# B&R Automation Studio project Palletizer
Automation Studio 4.10.2.37; technology packages: Acp10Arnc0 5.20.2, mappView 5.20.0

## Configuration Default_Config

CPU X20CP1382, AutomationRuntime A4.83, Build 4.1.2, Safety 0.0, Vc V4.72.3

### Hardware
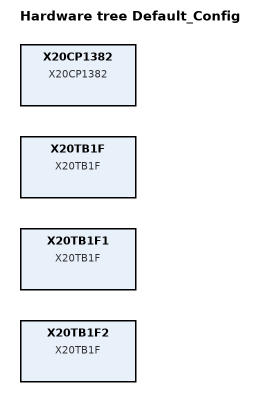
```
X20CP1382 : X20CP1382 v1.14.0.0  [X1 -> X1.SL; X2 -> X2.SL; X3 -> X3.SL]
  Module X1 (Type=X1, Virtual=true, Version=1.14.0.0)
    Connection (Connector=SS1, TargetModule=X20TB1F, TargetConnector=SS)
    Connection (Connector=SL, TargetModule=X20CP1382, TargetConnector=X1)
  Module X2 (Type=X2, Virtual=true, Version=1.14.0.0)
    Connection (Connector=SS1, TargetModule=X20TB1F1, TargetConnector=SS)
    Connection (Connector=SL, TargetModule=X20CP1382, TargetConnector=X2)
  Module X3 (Type=X3, Virtual=true, Version=1.14.0.0)
    Connection (Connector=SS1, TargetModule=X20TB1F2, TargetConnector=SS)
    Connection (Connector=SL, TargetModule=X20CP1382, TargetConnector=X3)
  Connector IF2:
    ActivateDevice = 1
    Vnc1
    VncKeyMappingFile1 = 
    VncRefreshRate1 = 100
  Connector IF3:
    DNAConfiguration = manual
    CycleTime = 2000
  ConfigurationID = Palletizer_Default_Config
  Simulation = 1
  Cyclic1Tolerance = 0
  Cyclic2Tolerance = 0
  TimeZone = 140
  ActivateOpcUa = 1
  OpcUaInformationModels_PV_Version = 1
X20TB1F : X20TB1F v1.0.0.0
X20TB1F1 : X20TB1F v1.0.0.0
X20TB1F2 : X20TB1F v1.0.0.0
```

### Acp10cfg.ncc - X20CP1382/Motion/Acp10cfg.ncc
```
NcConfiguration (Version=5.06.2, NcSwId=Acp10)
  ACP10CF1_typ:
    cnt_nettrc_rec_drive = 150
    bufsize_trace_upload = 1200
    tc_nc_man_task = Cyclic #1
    glob_pv_as_ncobject = Yes
    ncsys_dl_broadcast = Yes
    ncsys_dl_acp_reset = Yes
    safemc_log_err_to_ax = Yes
    network_init:
      ncsw_init_execute = Yes
      automatic_execute = No
      node_nr_warning = Yes
      net_err_before_ncact = Yes
    nettrc:
      enter_parsecrec = Yes
      enter_ncaction = Yes
      save_ring_startidx = No
    cam_prof_download:
      cam_dat_dl_parallel = No
      tc_cam_dl_parallel = Task class for NC Manager task
```

## Logical view

Binary libraries used (declarations not repeated): operator, runtime, astime, AsIecCon, standard, AsArLog, AsBrStr, AsTCP, MTBasics 2.21.0, brsystem, MTTypes 1.03.4, sys_lib, Acp10man 5.20.2, Acp10par 5.20.2, NcGlobal 5.20.2, Acp10sim 5.20.2

### Global.var - Global variables
```iecst
(*Sensors*)
VAR
	LightBarrier1 : BOOL;
	LightBarrier2 : BOOL;
	LaserSensor1 : BOOL;
	LaserSensor2 : BOOL;
END_VAR
(*Simulation variables*)
VAR
	Pusher_BKW : BOOL;
	Pusher_FWD : BOOL;
	Turnpusher_FWD : BOOL;
	Turnpusher_BWD : BOOL;
	Crane_Vacuum : BOOL;
	Pallet_ForkFB : BOOL;
	Feeder_ConveyorIF_Fwd : BOOL;
	Feeder_ConveyorTurn1_Fwd : BOOL;
	Feeder_PusherFwd : BOOL;
	Feeder_ConveyorEndFwd : BOOL;
	Feeder_TurnpusherFwd : BOOL;
	Feeder_TurnpusherBwd : BOOL;
	Crane_VacuumGrip : BOOL;
	Crane_CartboardTrig : BOOL;
	Crane_SlideRail_EN : BOOL;
	Crane_PusherZ_EN : BOOL;
	Crane_PusherX_EN : BOOL;
	Pallet_Fork_EN : BOOL;
	Pallet_Conveyor1_Fwd : BOOL;
	Feeder_Carriage_Axis : REAL;
	Feeder_Carriage_Reached : BOOL;
	Crane_Box_Axis : REAL;
	Crane_Gantry_Axis : REAL;
	Pallet_Lifter_Axis : REAL;
	Crane_Box_Axis_TgtPos : REAL;
	Feeder_Carriage_Axis_TgtPos : REAL;
	Crane_Gantry_Axis_TgtPos : REAL;
	Pallet_Conveyor2_ActVel : REAL;
	Pallet_Lifter_Axis_TgtPos : REAL;
END_VAR
(*Variables*)
VAR
	OperationType : INT := 0;
END_VAR
(*Faults*)
VAR
	OutOfPallet : BOOL;
	OutOfCartboard : BOOL;
	EmergencyStop : BOOL;
	Feeder_EmergencyStop : BOOL := FALSE;
	Crane_EmergencyStop : BOOL := FALSE;
	Pallet_EmergencyStop : BOOL := FALSE;
	Feeder_ResetConfig : BOOL := FALSE;
	Crane_ResetConfig : BOOL := FALSE;
	Pallet_ResetConfig : BOOL := FALSE;
	EnableMachine : BOOL := FALSE;
	Feeder_ImmediateStop : BOOL;
	Crane_ImmediateStop : BOOL;
	Pallet_ImmediateStop : BOOL;
	Feeder_Restart : BOOL := FALSE;
	Crane_Restart : BOOL := FALSE;
	Pallet_Restart : BOOL := FALSE;
	Feeder_OnPhaseStop : BOOL := FALSE;
	Crane_OnPhaseStop : BOOL := FALSE;
	Pallet_OnPhaseStop : BOOL := FALSE;
	ImmediateStop : BOOL;
	OnPhaseStop : BOOL;
	act_PalletConveyor2Fault : BOOL := FALSE;
	act_CartboardFault : BOOL := FALSE;
	act_CarriageFault : BOOL := FALSE;
	act_GantryCraneFault : BOOL := FALSE;
	act_BoxCraneFault : BOOL := FALSE;
	act_PalletForkFault : BOOL := FALSE;
	act_PalletLifterFault : BOOL := FALSE;
	act_FeederPusherFault : BOOL := FALSE;
	act_PusherXFault : BOOL := FALSE;
	act_PusherZFault : BOOL := FALSE;
	act_TurnpusherFault : BOOL := FALSE;
	act_SlideRailFault : BOOL := FALSE;
	act_ConveyorIFFault : BOOL := FALSE;
	act_ConveyorEndFault : BOOL := FALSE;
	act_PalletConveyor1Fault : BOOL := FALSE;
	act_ConveyorTurn1Fault : BOOL := FALSE;
	act_VacuumFault : BOOL := FALSE;
END_VAR
(*GenericDevices*)
VAR
	Conveyor_if_enable_request : BOOL;
	Conveyor_if_disable_request : BOOL;
	Conveyor_turn1_enable_request : BOOL;
	Conveyor_turn1_disable_request : BOOL;
	Pusher_enable_request : BOOL;
	Pusher_disable_request : BOOL;
	Conveyor_end_enable_request : BOOL;
	Conveyor_end_disable_request : BOOL;
	Turnpusher_enable_request : BOOL;
	Turnpusher_disable_request : BOOL;
	Vacuum_enable_request : BOOL;
	Vacuum_disable_request : BOOL;
	Cartboard_enable_request : BOOL;
	Cartboard_disable_request : BOOL;
	SlideRail_enable_request : BOOL;
	SlideRail_disable_request : BOOL;
	PusherZ_enable_request : BOOL;
	PusherZ_disable_request : BOOL;
	PusherX_enable_request : BOOL;
	PusherX_disable_request : BOOL;
	PalletFork_enable_request : BOOL;
	PalletFork_disable_request : BOOL;
	PalletConveyor1_enable_request : BOOL;
	PalletConveyor1_disable_request : BOOL;
END_VAR
(*Comunication between PALLET HANDLER and MAIN*)
VAR
	StartPallet : BOOL := FALSE; (*if TRUE the pallet handler goes to the idle state, ready to free a pallet*)
	PalletCounter : INT := 5; (*Number of pallets that are still available before a refill*)
END_VAR
(*Comunication between CRANE HANDLER and MAIN*)
VAR
	StartCrane : BOOL := FALSE; (*if TRUE the crane handler goes to the idle state, ready to receive the box layer*)
	CraneCartboardCounter : INT := 28;
END_VAR
(*Comunication between FEEDER_HANDLER and MAIN*)
VAR
	StartFeeder : BOOL := FALSE;
	CraneLayerCounter : BOOL := FALSE; (*If TRUE the feeder is working on the second layer*)
	BoxCounter : INT := 0;
END_VAR
(*MAIN*)
VAR
	StartMachine : BOOL; (*if TRUE the machine stars*)
	CraneReady : BOOL; (*if TRUE the crane is ready to receive the boxes*)
	FeederReady : BOOL; (*if TRUE the 14 boxes are ready to be loaded on the crane*)
	LoadBoxesOnCrane : BOOL; (*if TRUE the boxes can be loaded on the crane by the feeder*)
	BoxesOnCrane : BOOL; (*if TRUE the boxes are ready to be held by the crane*)
	HoldBoxes : BOOL; (*if TRUE boxes are held by the crane*)
	PalletReady : BOOL; (*if TRUE the pallet is in position*)
	LoadBoxesOnPallet : BOOL; (*if TRUE the boxes will be loaded on the pallet*)
	SecondLayer : BOOL; (*if TRUE the feeder has finished the second layer*)
	BoxesOnPallet : BOOL; (*if TRUE the boxes are on the pallet*)
	PalletExit_EN : BOOL; (*if TRUE the pallet can move to the next station*)
	PalletExit_DONE : BOOL; (*if TRUE the pallet has gone to the next station*)
	SIMConveyorIFFault : BOOL := FALSE;
	SIMConveyorTurn1Fault : BOOL := FALSE;
	SIMFeederPusherFault : BOOL := FALSE;
	SIMConveyorEndFault : BOOL := FALSE;
	SIMTurnpusherFault : BOOL := FALSE;
	SIMCarriageFault : BOOL := FALSE;
	SIMVacuumFault : BOOL := FALSE;
	SIMSlideRailFault : BOOL := FALSE;
	SIMPusherZFault : BOOL := FALSE;
	SIMPusherXFault : BOOL := FALSE;
	SIMGantryCraneFault : BOOL := FALSE;
	SIMBoxCraneFault : BOOL := FALSE;
	SIMPalletForkFault : BOOL := FALSE;
	SIMPalletConveyor1Fault : BOOL := FALSE;
	SIMPalletLifterFault : BOOL := FALSE;
	SIMCartboardFault : BOOL := FALSE;
	SIMPalletConveyor2Fault : BOOL := FALSE;
END_VAR
(**)
VAR
	OutOfMaterial : BOOL;
END_VAR
```

### MNG_Global.typ - Global data types
```iecst
(* 3d position *)
(* position and orientation as an euler based pose *)
(* position and orientation as a 4x4 matrix *)

TYPE
	VEC3 : 	STRUCT
		x : REAL;
		y : REAL;
		z : REAL;
	END_STRUCT;
	POSE6 : 	STRUCT
		x : REAL;
		y : REAL;
		z : REAL;
		a : REAL;
		b : REAL;
		c : REAL;
	END_STRUCT;
	TRAFO : 	STRUCT
		baseX : VEC3;
		fill0 : REAL;
		baseY : VEC3;
		fill1 : REAL;
		baseZ : VEC3;
		fill2 : REAL;
		origin : VEC3;
		fill3 : REAL;
	END_STRUCT;
END_TYPE
```

### MNG_Package.typ
```iecst
(*                                                                            *)
(* File generated by the B&R AS 4 control config generator                    *)
(*                                                                            *)
(*     Provider: machineering                                                 *)
(*  Application: industrialPhysics_2.4.master                                 *)
(* Architecture: Windows 64 Bit                                               *)
(*      Version: 2.4.10491.master                                             *)
(*        Build: 164f85bec                                                    *)
(*         Date: 2020-05-19, Time: 12:11:21                                   *)
(*                                                                            *)

TYPE
	ComTCP_INPUTS_32BIT : 	STRUCT
		NumSignals : INT := 15;
		laser_sensor_IR : BOOL := 0; (* BOOL laser_sensor_IR *)
		laser_sensor2_IR : BOOL := 0; (* BOOL laser_sensor2_IR *)
		carriage_2_AXIS : REAL := 0.0; (* REAL carriage_2_AXIS *)
		carriage_2_RCHD : BOOL := 0; (* BOOL carriage_2_RCHD *)
		turnpusher_LBK : BOOL := 0; (* BOOL turnpusher_LBK *)
		turnpusher_LFR : BOOL := 0; (* BOOL turnpusher_LFR *)
		gantry_crane_AXIS : REAL := 0.0; (* REAL gantry_crane_AXIS *)
		box_crane_AXIS : REAL := 0.0; (* REAL box_crane_AXIS *)
		vaccum_box_crane_VACUUM : BOOL := 0; (* BOOL vaccum_box_crane_VACUUM *)
		pallet_light_barrier_1_IR : BOOL := 0; (* BOOL pallet_light_barrier_1_IR *)
		pallet_light_barrier_2_IR : BOOL := 0; (* BOOL pallet_light_barrier_2_IR *)
		pusher_LBK : BOOL := 0; (* BOOL pusher_LBK *)
		pusher_LFR : BOOL := 0; (* BOOL pusher_LFR *)
		pallet_lifter_AXIS : REAL := 0.0; (* REAL pallet_lifter_AXIS *)
		pallet_fork_left_FB : BOOL := 0; (* BOOL pallet_fork_left_FB *)
	END_STRUCT;
	ComTCP_OUTPUTS_32BIT : 	STRUCT
		NumSignals : INT := 18;
		cartboard_TRIG : BOOL := 0; (* BOOL cartboard_TRIG *)
		conveyor_if_FWD : BOOL := 0; (* BOOL conveyor_if_FWD *)
		conveyer_turn1_FWD : BOOL := 0; (* BOOL conveyer_turn1_FWD *)
		conveyer_end_FWD : BOOL := 0; (* BOOL conveyer_end_FWD *)
		carriage_2_TGT_POS : REAL := 0.0; (* REAL carriage_2_TGT_POS *)
		turnpusher_FWD : BOOL := 0; (* BOOL turnpusher_FWD *)
		turnpusher_BWD : BOOL := 0; (* BOOL turnpusher_BWD *)
		gantry_crane_TGT_POS : REAL := 0.0; (* REAL gantry_crane_TGT_POS *)
		box_crane_TGT_POS : REAL := 0.0; (* REAL box_crane_TGT_POS *)
		slide_rail_right_EN : BOOL := 0; (* BOOL slide_rail_right_EN *)
		vaccum_box_crane_GRIP : BOOL := 0; (* BOOL vaccum_box_crane_GRIP *)
		pusher_z_EN : BOOL := 0; (* BOOL pusher_z_EN *)
		pusher_x_EN : BOOL := 0; (* BOOL pusher_x_EN *)
		pallet_conveyor_2_ACT_VEL : REAL := 0.0; (* REAL pallet_conveyor_2_ACT_VEL *)
		pusher_FW : BOOL := 0; (* BOOL pusher_FW *)
		pallet_lifter_TGT_POS : REAL := 0.0; (* REAL pallet_lifter_TGT_POS *)
		pallet_fork_left_EN : BOOL := 0; (* BOOL pallet_fork_left_EN *)
		pallet_conveyor_1_FWD : BOOL := 0; (* BOOL pallet_conveyor_1_FWD *)
	END_STRUCT;
END_TYPE
```

### MNG_Package.var
```iecst
(*                                                                            *)
(* File generated by the B&R AS 4 control config generator                    *)
(*                                                                            *)
(*     Provider: machineering                                                 *)
(*  Application: industrialPhysics_2.4.master                                 *)
(* Architecture: Windows 64 Bit                                               *)
(*      Version: 2.4.10491.master                                             *)
(*        Build: 164f85bec                                                    *)
(*         Date: 2020-05-19, Time: 12:11:21                                   *)
(*                                                                            *)
VAR
	ComTCP_SimInputs : ComTCP_INPUTS_32BIT := (0);
	ComTCP_SimOutputs : ComTCP_OUTPUTS_32BIT := (0);
	ComTCP_SimServerAddress : STRING[15] := '127.0.0.1';
	ComTCP_SimServerPort : UINT := 5000;
	ComTCP_SimSendCycleTime : TIME := T#5ms;
	ComTCP_SimActive : BOOL := FALSE;
END_VAR
```

### Package Logical/Libraries - Global libraries

### Library Logical/Libraries/ComTCP/ComTCP_L (ANSIC)
Depends on: AsTCP, operator, runtime, astime, standard, AsArLog, AsBrStr, Convert

#### MNG_InternalTyp.hpp
```cpp
#ifndef _MNGINTERNALTYP_HPP_
#define _MNGINTERNALTYP_HPP_

#include <AsIecCon.h>
#include <AsBrStr.h>

#include "MNG_Global.hpp"

typedef enum {
	MNG_DeadManDatagram = 0,
	MNG_TimeTick,
	MNG_TimeTickRequest,
	MNG_InitConnection,
	MNG_ResetSimulation,
	MNG_RewindSimulation,
	MNG_StartSimulation,
	MNG_StopSimulation,
	MNG_IOConfig,
	MNG_RawIOImage,
	MNG_Raw32BitImage,
	MNG_TextDatagram,
	MNG_UnknownDatagram
}MNG_DatagramType;

typedef struct {
	unsigned long int Counter;
	unsigned long int SentTime;
	unsigned long int DatagramType;
	unsigned long int ByteCount;
}MNG_DatagramHeader;

typedef unsigned long int MNG_DataArray[1400];

typedef struct {
	MNG_DatagramHeader Header;
	MNG_DataArray Payload;
}MNG_RawDatagram;

#endif
```

#### MNG_ComHdlr.hpp
```cpp
#ifndef _MNGCOMHDLR_HPP_
#define _MNGCOMHDLR_HPP_

#define TRUE  1
#define FALSE 0

#include "MNG_InternalTyp.hpp"

#include <bur/plc.h>
#include <bur/plctypes.h>
#include <AsTCP.h>
#include <standard.h>
#include <astime.h>
#include <runtime.h>
#include <AsBrStr.h>

typedef struct{
	TcpOpen_typ tcpOpen;
	TcpIoctl_typ tcpIoctl;
	tcpLINGER_typ tcpLINGER;
	TcpSend_typ tcpSend;
	TcpClose_typ tcpClose;
	TcpRecv_typ tcpRecv;
	TcpClient_typ tcpClient;
} asTcpFcn_t;

typedef enum {
	MNG_wSock,
	MNG_skippedMessage
} MNG_errorCases;

typedef enum {
	MNG_Init,
	MNG_Socket,
	MNG_Open,
	MNG_SetIo,
	MNG_Linger,
	MNG_Connecting,
	MNG_Exchange,
	MNG_Closing,
        MNG_Reset
} MNG_internalState_t;

	extern unsigned long int MNG_CpyOutToMsg(MNG_RawDatagram * pToServer, unsigned long int counter, ComTCP_OUTPUTS_32BIT_FWRD *pSimOutputs);
	extern unsigned long int MNG_CpyMsgToInp(MNG_RawDatagram * pFromServer, ComTCP_INPUTS_32BIT_FWRD *pSimInputs);

class MNG_ComHdlr
{
	public:

	MNG_ComHdlr(char *srvIpAdr, unsigned int srvPort, TIME sendCycleTime);
	~MNG_ComHdlr();

        int RunCommunication(void*, void*, BOOL*);

	private:

	char* _srvIpAdr;
	unsigned int _srvPort;
	TIME _sendCycleTime;

	unsigned int _error;

	MNG_internalState_t _internalState;
	TON_typ _connectionTon;
	TIME _connectionTime;

	bool _connect;
	bool _sendDone;

	signed int _recvOffset;

	signed long int _potMsgLen;
	signed long int _totalRecvLen;

	unsigned long int _one;
	unsigned long int _counter;
	unsigned long int _recvLen;
	unsigned long int _recvBuffer[10000];
	TON_typ _sendTon;
	MNG_RawDatagram _recvMessage;
	MNG_RawDatagram _sendMessage;

	static const signed long int SIXTEEN = 16;
	static const unsigned int PORT = 0;
	static const unsigned long int MNG_MAXPAYLOAD = 1400;

	void init_TcpOpen();
	void init_TcpSocket();
	void init_TcpIoctl();
	void init_TcpLinger();
	void init_TcpClient();
	void init_TcpRecv();
	void init_TcpSend(ComTCP_OUTPUTS_32BIT_FWRD* pSimOut);

	void InitParams();

	void SetSendDone(bool toogle);
	void SetStateValue(MNG_internalState_t stateVal);

};
#endif
```

#### MNG_ComHdlr.cpp
```cpp
#include "MNG_ComHdlr.hpp"
#include "MNG_CpyMsgToInp.cpp"
#include "MNG_CpyOutToMsg.cpp"

asTcpFcn_t _asTcpFcn;

MNG_ComHdlr::MNG_ComHdlr(char *srvIpAdr, unsigned int srvPort, TIME sendCycleTime)
{
	_srvIpAdr = srvIpAdr;
	_srvPort = srvPort;
	_sendCycleTime = sendCycleTime;
	InitParams();
}

MNG_ComHdlr::~MNG_ComHdlr()
{
}

int MNG_ComHdlr::RunCommunication(void* pSimInputs, void* pSimOutputs, BOOL* pSimActive) {

        unsigned long int _lastCounter = _counter;

	ComTCP_INPUTS_32BIT_FWRD* pFwrd_SimInputs = static_cast<ComTCP_INPUTS_32BIT_FWRD*>((pSimInputs));
	ComTCP_OUTPUTS_32BIT_FWRD* pFwrd_SimOutputs = static_cast<ComTCP_OUTPUTS_32BIT_FWRD*>((pSimOutputs));

	switch (_internalState) {

		case MNG_Init:
                        *pSimActive = FALSE;
			_asTcpFcn.tcpOpen.enable = FALSE;
			TcpOpen(&_asTcpFcn.tcpOpen);
			_asTcpFcn.tcpIoctl.enable = FALSE;
			TcpIoctl(&_asTcpFcn.tcpIoctl);
			_asTcpFcn.tcpClient.enable = FALSE;
			TcpClient(&_asTcpFcn.tcpClient);
			_asTcpFcn.tcpSend.enable = FALSE;
			TcpSend(&_asTcpFcn.tcpSend);
			_asTcpFcn.tcpRecv.enable = FALSE;
			TcpRecv(&_asTcpFcn.tcpRecv);
			_asTcpFcn.tcpClose.enable = FALSE;
			TcpClose(&_asTcpFcn.tcpClose);

			_connectionTon.IN = FALSE;
			_connectionTon.PT = _connectionTime;
			_sendTon.IN = FALSE;
			_sendTon.PT = _sendCycleTime;
			SetStateValue(MNG_Socket);
			break;

		case MNG_Socket:
                        *pSimActive = FALSE;
			init_TcpSocket();
			TcpOpen(&_asTcpFcn.tcpOpen);
			_recvOffset = 0;
			if (_connect == 1) {
				SetStateValue(MNG_Open);
				_connectionTon.IN = FALSE;
			}
			break;

		case MNG_Open:
                        *pSimActive = FALSE;
			init_TcpOpen();
			TcpOpen(&_asTcpFcn.tcpOpen);
			if (_asTcpFcn.tcpOpen.status == 0) {
				SetStateValue(MNG_SetIo);
				_asTcpFcn.tcpIoctl.enable = FALSE;
				TcpIoctl(&_asTcpFcn.tcpIoctl);
				_connectionTon.IN = FALSE;
			}
			break;

		case MNG_SetIo:
                        *pSimActive = FALSE;
			init_TcpIoctl();
			TcpIoctl(&_asTcpFcn.tcpIoctl);
			if (_asTcpFcn.tcpIoctl.status == 0) {
				SetStateValue(MNG_Linger);
				_asTcpFcn.tcpClient.enable = FALSE;
				TcpClient(&_asTcpFcn.tcpClient);
				_connectionTon.IN = FALSE;
			}
			break;

		case MNG_Linger:
                        *pSimActive = FALSE;
			init_TcpLinger();
			TcpIoctl(&_asTcpFcn.tcpIoctl);

			if (_asTcpFcn.tcpIoctl.status == 0) {
				SetStateValue(MNG_Connecting);
				_asTcpFcn.tcpClient.enable = FALSE;
				_connectionTon.IN = FALSE;
			}

		case MNG_Connecting:
                        *pSimActive = FALSE;
			_asTcpFcn.tcpClient.enable = TRUE;
			_asTcpFcn.tcpClient.ident = _asTcpFcn.tcpOpen.ident;
			_asTcpFcn.tcpClient.portserv = _srvPort;
			_asTcpFcn.tcpClient.pServer = (long)_srvIpAdr;
			TcpClient(&_asTcpFcn.tcpClient);

			if (_asTcpFcn.tcpClient.status == ERR_FUB_BUSY) {
				// state = state || SetStateValue(Connecting);
			} else if (_asTcpFcn.tcpClient.status == 0) {
				SetStateValue(MNG_Exchange);
				_connectionTon.IN = FALSE;
				SetSendDone(TRUE);
			}
			break;

		case MNG_Exchange:
			init_TcpRecv();
			TcpRecv(&_asTcpFcn.tcpRecv);

			if (_asTcpFcn.tcpRecv.status==0){
                        *pSimActive = FALSE;
			_connectionTon.IN = FALSE;
			_recvLen = _asTcpFcn.tcpRecv.recvlen;
			_potMsgLen = N_TO_HUDINT(_recvBuffer[3]) + SIXTEEN;
			_totalRecvLen = _recvOffset + _recvLen;

			if ((_totalRecvLen < SIXTEEN) || (_totalRecvLen < _potMsgLen)) {
			_recvOffset = _recvOffset + _recvLen;
			}	else {
			while ((_potMsgLen > 0) && (_potMsgLen <= _totalRecvLen)) {
			// misconfigured message sizes
                        if ((unsigned long int)_potMsgLen > sizeof(_recvMessage)) {
			SetStateValue(MNG_Reset);
			break;
			}

			brsmemcpy((unsigned long int) &_recvMessage, (unsigned long int) &_recvBuffer, _potMsgLen*sizeof(unsigned long int));
			_totalRecvLen = _totalRecvLen - _potMsgLen;
			brsmemmove((unsigned long int) &_recvBuffer, (unsigned long int) &_recvBuffer + _potMsgLen, _totalRecvLen*sizeof(unsigned long int));
			_counter = MNG_CpyMsgToInp(&_recvMessage,pFwrd_SimInputs);
                        *pSimActive = (_lastCounter != _counter);
			_recvOffset = _totalRecvLen;

			if (_totalRecvLen > SIXTEEN) {
			_potMsgLen = N_TO_HUDINT(_recvBuffer[3]) + SIXTEEN;
			} else {
			_potMsgLen = 0;
			}

			}
			}
			}

			_sendTon.IN = _sendDone;
			TON(&_sendTon);

			if (_sendTon.Q || _asTcpFcn.tcpSend.enable == 1) {
				if (_sendDone==TRUE) {
					SetSendDone(FALSE);
					MNG_CpyOutToMsg(&_sendMessage, _counter,pFwrd_SimOutputs);
					init_TcpSend(pFwrd_SimOutputs);
				}
				TcpSend(&_asTcpFcn.tcpSend);

				if (_asTcpFcn.tcpSend.status == 0) {
					if (_asTcpFcn.tcpSend.datalen != _asTcpFcn.tcpSend.sentlen) {
						// state = state || SetStateValue(Exchange);
					}
					_asTcpFcn.tcpSend.enable = FALSE;
					SetSendDone(TRUE);
				}
			}
			if (_asTcpFcn.tcpRecv.status == tcpERR_NOT_CONNECTED) {
				SetStateValue(MNG_Closing);
			}
			break;

		case MNG_Closing:
                        *pSimActive = FALSE;
			_asTcpFcn.tcpClose.enable = TRUE;
			_asTcpFcn.tcpClose.ident = _asTcpFcn.tcpOpen.ident;
			_asTcpFcn.tcpClose.how = 0;
			TcpClose(&_asTcpFcn.tcpClose);

			if(_asTcpFcn.tcpClose.status == 0 || _asTcpFcn.tcpClose.status == 32600){
				SetStateValue(MNG_Init);
			}
			break;

                case MNG_Reset:
                        SetStateValue(MNG_Closing);
                        break;
	}

	TON(&_connectionTon);
	_connectionTon.IN = TRUE;
	if (_connectionTon.Q == 1) {
		SetStateValue(MNG_Closing);
		_connectionTon.IN = FALSE;
	}

	return _internalState;
}

void MNG_ComHdlr::init_TcpOpen(){
	_asTcpFcn.tcpOpen.enable = _connect;
}

void MNG_ComHdlr::init_TcpSocket(){
	_asTcpFcn.tcpOpen.enable = TRUE;
	_asTcpFcn.tcpOpen.pIfAddr = 0;
	_asTcpFcn.tcpOpen.port = PORT;
	_asTcpFcn.tcpOpen.options = tcpOPT_REUSEADDR;
}

void MNG_ComHdlr::init_TcpIoctl(){
	_asTcpFcn.tcpIoctl.enable = TRUE;
	_asTcpFcn.tcpIoctl.pData = (unsigned long int) &_one;
	_asTcpFcn.tcpIoctl.datalen = 4;
	_asTcpFcn.tcpIoctl.ident = _asTcpFcn.tcpOpen.ident;
	_asTcpFcn.tcpIoctl.ioctl = tcpTCP_NODELAY_SET;
}

void MNG_ComHdlr::init_TcpLinger(){
	_asTcpFcn.tcpLINGER.lLinger = FALSE;
	_asTcpFcn.tcpLINGER.lOnOff = TRUE;
	_asTcpFcn.tcpIoctl.enable = TRUE;
	_asTcpFcn.tcpIoctl.pData = (unsigned long int) &_asTcpFcn.tcpLINGER;
	_asTcpFcn.tcpIoctl.datalen = sizeof(_asTcpFcn.tcpLINGER);
	_asTcpFcn.tcpIoctl.ident = _asTcpFcn.tcpOpen.ident;
	_asTcpFcn.tcpIoctl.ioctl = tcpSO_LINGER_SET;
}

void MNG_ComHdlr::init_TcpClient(){

	_asTcpFcn.tcpClient.enable = TRUE;
	_asTcpFcn.tcpClient.ident = _asTcpFcn.tcpOpen.ident;
	_asTcpFcn.tcpClient.portserv = _srvPort;
	_asTcpFcn.tcpClient.pServer = (long)_srvIpAdr;
}

void MNG_ComHdlr::init_TcpRecv(){

	_asTcpFcn.tcpRecv.enable = TRUE;
	_asTcpFcn.tcpRecv.ident= _asTcpFcn.tcpOpen.ident;
	_asTcpFcn.tcpRecv.datamax = sizeof(_recvBuffer) - _recvOffset;
	_asTcpFcn.tcpRecv.pData = (unsigned long int) &_recvBuffer + _recvOffset;
}

void MNG_ComHdlr::init_TcpSend(ComTCP_OUTPUTS_32BIT_FWRD *pSimOutputs){

	_asTcpFcn.tcpSend.enable = TRUE;
	_asTcpFcn.tcpSend.ident= _asTcpFcn.tcpOpen.ident;
	_asTcpFcn.tcpSend.datalen = 16 + ((pSimOutputs->NumSignals) + 1) * 4;
	_asTcpFcn.tcpSend.pData = (unsigned long int)&_sendMessage;
	_asTcpFcn.tcpSend.flags = 0;
}

void MNG_ComHdlr::InitParams(){
	_internalState = MNG_Init;
	_connectionTime = 3000;
	_one=1;
	_connect = TRUE;
	_potMsgLen = 0;
	_recvLen = 0;
	_recvOffset = 0;
	_counter = 0;
	SetSendDone(FALSE);
}

void MNG_ComHdlr::SetSendDone(bool toggle){
	_sendDone=toggle;
}

void MNG_ComHdlr::SetStateValue(MNG_internalState_t stateVal){
	_internalState=stateVal;
}
```

#### MNG_Global.hpp
```cpp
#ifndef  _MNGGLOBAL_HPP_
#define _MNGGLOBAL_HPP_

#include <mng_globalTYP.h>

    typedef struct {

		signed short NumSignals;

        /* BOOL laser_sensor_IR */
        BOOL laser_sensor_IR;
        /* BOOL laser_sensor2_IR */
        BOOL laser_sensor2_IR;
        /* REAL carriage_2_AXIS */
        REAL carriage_2_AXIS;
        /* BOOL carriage_2_RCHD */
        BOOL carriage_2_RCHD;
        /* BOOL turnpusher_LBK */
        BOOL turnpusher_LBK;
        /* BOOL turnpusher_LFR */
        BOOL turnpusher_LFR;
        /* REAL gantry_crane_AXIS */
        REAL gantry_crane_AXIS;
        /* REAL box_crane_AXIS */
        REAL box_crane_AXIS;
        /* BOOL vaccum_box_crane_VACUUM */
        BOOL vaccum_box_crane_VACUUM;
        /* BOOL pallet_light_barrier_1_IR */
        BOOL pallet_light_barrier_1_IR;
        /* BOOL pallet_light_barrier_2_IR */
        BOOL pallet_light_barrier_2_IR;
        /* BOOL pusher_LBK */
        BOOL pusher_LBK;
        /* BOOL pusher_LFR */
        BOOL pusher_LFR;
        /* REAL pallet_lifter_AXIS */
        REAL pallet_lifter_AXIS;
        /* BOOL pallet_fork_left_FB */
        BOOL pallet_fork_left_FB;

        } ComTCP_INPUTS_32BIT_FWRD;

    typedef struct {

		signed short NumSignals;

        /* BOOL cartboard_TRIG */
        BOOL cartboard_TRIG;
        /* BOOL conveyor_if_FWD */
        BOOL conveyor_if_FWD;
        /* BOOL conveyer_turn1_FWD */
        BOOL conveyer_turn1_FWD;
        /* BOOL conveyer_end_FWD */
        BOOL conveyer_end_FWD;
        /* REAL carriage_2_TGT_POS */
        REAL carriage_2_TGT_POS;
        /* BOOL turnpusher_FWD */
        BOOL turnpusher_FWD;
        /* BOOL turnpusher_BWD */
        BOOL turnpusher_BWD;
        /* REAL gantry_crane_TGT_POS */
        REAL gantry_crane_TGT_POS;
        /* REAL box_crane_TGT_POS */
        REAL box_crane_TGT_POS;
        /* BOOL slide_rail_right_EN */
        BOOL slide_rail_right_EN;
        /* BOOL vaccum_box_crane_GRIP */
        BOOL vaccum_box_crane_GRIP;
        /* BOOL pusher_z_EN */
        BOOL pusher_z_EN;
        /* BOOL pusher_x_EN */
        BOOL pusher_x_EN;
        /* REAL pallet_conveyor_2_ACT_VEL */
        REAL pallet_conveyor_2_ACT_VEL;
        /* BOOL pusher_FW */
        BOOL pusher_FW;
        /* REAL pallet_lifter_TGT_POS */
        REAL pallet_lifter_TGT_POS;
        /* BOOL pallet_fork_left_EN */
        BOOL pallet_fork_left_EN;
        /* BOOL pallet_conveyor_1_FWD */
        BOOL pallet_conveyor_1_FWD;

        } ComTCP_OUTPUTS_32BIT_FWRD;

#endif
```

#### MNG_CpyOutToMsg.cpp
```cpp
#include "MNG_InternalTyp.hpp"

unsigned long int MNG_CpyOutToMsg(MNG_RawDatagram * pToServer, unsigned long int counter, ComTCP_OUTPUTS_32BIT_FWRD *pSimOutputs ) {

        unsigned long int DWordBuffer;

        pSimOutputs->NumSignals = 18;
        (pToServer->Header).ByteCount    = H_TO_NUDINT(76);
        (pToServer->Header).DatagramType = H_TO_NUDINT(MNG_Raw32BitImage);
        (pToServer->Header).SentTime = H_TO_NUDINT(0);  // Todo
        (pToServer->Header).Counter = H_TO_NUDINT(counter);
        pToServer->Payload[0] = H_TO_NUDINT(pSimOutputs->NumSignals);

    /* cartboard_TRIG : BOOL */
    if(pSimOutputs->cartboard_TRIG == 1) {
        pToServer->Payload[1] = 0xFFFFFFFF;   /*BOOL */
    } else {
        pToServer->Payload[1] = 0;
    }

    /* conveyor_if_FWD : BOOL */
    if(pSimOutputs->conveyor_if_FWD == 1) {
        pToServer->Payload[2] = 0xFFFFFFFF;   /*BOOL */
    } else {
        pToServer->Payload[2] = 0;
    }

    /* conveyer_turn1_FWD : BOOL */
    if(pSimOutputs->conveyer_turn1_FWD == 1) {
        pToServer->Payload[3] = 0xFFFFFFFF;   /*BOOL */
    } else {
        pToServer->Payload[3] = 0;
    }

    /* conveyer_end_FWD : BOOL */
    if(pSimOutputs->conveyer_end_FWD == 1) {
        pToServer->Payload[4] = 0xFFFFFFFF;   /*BOOL */
    } else {
        pToServer->Payload[4] = 0;
    }

    /* carriage_2_TGT_POS : FLOAT32 */
    brsmemcpy((unsigned long int)&(DWordBuffer), (unsigned long int)&(pSimOutputs->carriage_2_TGT_POS), 4);
    pToServer->Payload[5] = H_TO_NUDINT(DWordBuffer);

    /* turnpusher_FWD : BOOL */
    if(pSimOutputs->turnpusher_FWD == 1) {
        pToServer->Payload[6] = 0xFFFFFFFF;   /*BOOL */
    } else {
        pToServer->Payload[6] = 0;
    }

    /* turnpusher_BWD : BOOL */
    if(pSimOutputs->turnpusher_BWD == 1) {
        pToServer->Payload[7] = 0xFFFFFFFF;   /*BOOL */
    } else {
        pToServer->Payload[7] = 0;
    }

    /* gantry_crane_TGT_POS : FLOAT32 */
    brsmemcpy((unsigned long int)&(DWordBuffer), (unsigned long int)&(pSimOutputs->gantry_crane_TGT_POS), 4);
    pToServer->Payload[8] = H_TO_NUDINT(DWordBuffer);

    /* box_crane_TGT_POS : FLOAT32 */
    brsmemcpy((unsigned long int)&(DWordBuffer), (unsigned long int)&(pSimOutputs->box_crane_TGT_POS), 4);
    pToServer->Payload[9] = H_TO_NUDINT(DWordBuffer);

    /* slide_rail_right_EN : BOOL */
    if(pSimOutputs->slide_rail_right_EN == 1) {
        pToServer->Payload[10] = 0xFFFFFFFF;   /*BOOL */
    } else {
        pToServer->Payload[10] = 0;
    }

    /* vaccum_box_crane_GRIP : BOOL */
    if(pSimOutputs->vaccum_box_crane_GRIP == 1) {
        pToServer->Payload[11] = 0xFFFFFFFF;   /*BOOL */
    } else {
        pToServer->Payload[11] = 0;
    }

    /* pusher_z_EN : BOOL */
    if(pSimOutputs->pusher_z_EN == 1) {
        pToServer->Payload[12] = 0xFFFFFFFF;   /*BOOL */
    } else {
        pToServer->Payload[12] = 0;
    }

    /* pusher_x_EN : BOOL */
    if(pSimOutputs->pusher_x_EN == 1) {
        pToServer->Payload[13] = 0xFFFFFFFF;   /*BOOL */
    } else {
        pToServer->Payload[13] = 0;
    }

    /* pallet_conveyor_2_ACT_VEL : FLOAT32 */
    brsmemcpy((unsigned long int)&(DWordBuffer), (unsigned long int)&(pSimOutputs->pallet_conveyor_2_ACT_VEL), 4);
    pToServer->Payload[14] = H_TO_NUDINT(DWordBuffer);

    /* pusher_FW : BOOL */
    if(pSimOutputs->pusher_FW == 1) {
        pToServer->Payload[15] = 0xFFFFFFFF;   /*BOOL */
    } else {
        pToServer->Payload[15] = 0;
    }

    /* pallet_lifter_TGT_POS : FLOAT32 */
    brsmemcpy((unsigned long int)&(DWordBuffer), (unsigned long int)&(pSimOutputs->pallet_lifter_TGT_POS), 4);
    pToServer->Payload[16] = H_TO_NUDINT(DWordBuffer);

    /* pallet_fork_left_EN : BOOL */
    if(pSimOutputs->pallet_fork_left_EN == 1) {
        pToServer->Payload[17] = 0xFFFFFFFF;   /*BOOL */
    } else {
        pToServer->Payload[17] = 0;
    }

    /* pallet_conveyor_1_FWD : BOOL */
    if(pSimOutputs->pallet_conveyor_1_FWD == 1) {
        pToServer->Payload[18] = 0xFFFFFFFF;   /*BOOL */
    } else {
        pToServer->Payload[18] = 0;
    }

	return 0;
}
```

#### MNG_CpyMsgToInp.cpp
```cpp
#include "MNG_InternalTyp.hpp"

unsigned long int MNG_CpyMsgToInp(MNG_RawDatagram * pFromServer, ComTCP_INPUTS_32BIT_FWRD *pSimInputs) {

    MNG_DatagramType datagramType;
	unsigned long int DWordBuffer;
        unsigned long int byteCount;
	unsigned long int numSignalsInMessage;

	byteCount = N_TO_HUDINT((pFromServer->Header).ByteCount);
	datagramType = static_cast<MNG_DatagramType>(N_TO_HUDINT((pFromServer->Header).DatagramType));
	if (datagramType != MNG_Raw32BitImage) {
		return 0;
	}

    pSimInputs->NumSignals = 15;

    numSignalsInMessage = N_TO_HUDINT(pFromServer->Payload[0]);
        if ((static_cast<long int>(numSignalsInMessage) != pSimInputs->NumSignals) ||
	(byteCount != 4 + numSignalsInMessage * 4)) {
		return 0;
	}

    /* BOOL laser_sensor_IR */
    pSimInputs->laser_sensor_IR = (pFromServer->Payload[1] != 0);

    /* BOOL laser_sensor2_IR */
    pSimInputs->laser_sensor2_IR = (pFromServer->Payload[2] != 0);

    /* FLOAT32 carriage_2_AXIS */
    DWordBuffer = N_TO_HUDINT(pFromServer->Payload[3]);
    brsmemcpy((unsigned long int)&(pSimInputs->carriage_2_AXIS), (unsigned long int)&(DWordBuffer), 4);

    /* BOOL carriage_2_RCHD */
    pSimInputs->carriage_2_RCHD = (pFromServer->Payload[4] != 0);

    /* BOOL turnpusher_LBK */
    pSimInputs->turnpusher_LBK = (pFromServer->Payload[5] != 0);

    /* BOOL turnpusher_LFR */
    pSimInputs->turnpusher_LFR = (pFromServer->Payload[6] != 0);

    /* FLOAT32 gantry_crane_AXIS */
    DWordBuffer = N_TO_HUDINT(pFromServer->Payload[7]);
    brsmemcpy((unsigned long int)&(pSimInputs->gantry_crane_AXIS), (unsigned long int)&(DWordBuffer), 4);

    /* FLOAT32 box_crane_AXIS */
    DWordBuffer = N_TO_HUDINT(pFromServer->Payload[8]);
    brsmemcpy((unsigned long int)&(pSimInputs->box_crane_AXIS), (unsigned long int)&(DWordBuffer), 4);

    /* BOOL vaccum_box_crane_VACUUM */
    pSimInputs->vaccum_box_crane_VACUUM = (pFromServer->Payload[9] != 0);

    /* BOOL pallet_light_barrier_1_IR */
    pSimInputs->pallet_light_barrier_1_IR = (pFromServer->Payload[10] != 0);

    /* BOOL pallet_light_barrier_2_IR */
    pSimInputs->pallet_light_barrier_2_IR = (pFromServer->Payload[11] != 0);

    /* BOOL pusher_LBK */
    pSimInputs->pusher_LBK = (pFromServer->Payload[12] != 0);

    /* BOOL pusher_LFR */
    pSimInputs->pusher_LFR = (pFromServer->Payload[13] != 0);

    /* FLOAT32 pallet_lifter_AXIS */
    DWordBuffer = N_TO_HUDINT(pFromServer->Payload[14]);
    brsmemcpy((unsigned long int)&(pSimInputs->pallet_lifter_AXIS), (unsigned long int)&(DWordBuffer), 4);

    /* BOOL pallet_fork_left_FB */
    pSimInputs->pallet_fork_left_FB = (pFromServer->Payload[15] != 0);

return N_TO_HUDINT((pFromServer->Header).Counter); // return counter
}
```

### Program Logical/Libraries/ComTCP/ComTCP_P (ANSIC)

#### Main.cpp - Init, cyclic, exit code
```cpp
#include <bur/plctypes.h>

#ifdef _DEFAULT_INCLUDES
        #include <AsDefault.h>
#endif

#include "../ComTCP_L/MNG_Global.hpp"
#include "../ComTCP_L/MNG_InternalTyp.hpp"
#include "../ComTCP_L/MNG_ComHdlr.hpp"

unsigned long bur_heap_size = 0xFFFF;

MNG_ComHdlr *pMNG_ComHdlr;

void _INIT ProgramInit(void)
{
    pMNG_ComHdlr = new MNG_ComHdlr(ComTCP_SimServerAddress, ComTCP_SimServerPort, ComTCP_SimSendCycleTime);
}

void _CYCLIC ProgramCyclic(void)
{
    connectionState = pMNG_ComHdlr->RunCommunication((void*)&ComTCP_SimInputs,(void*)&ComTCP_SimOutputs, &ComTCP_SimActive);
}

void _EXIT ProgramExit(void)
{
    delete pMNG_ComHdlr;
}
```

#### Variables.var - Local variables
```iecst
VAR
	connectionState : INT;
END_VAR
```

### Library Logical/Libraries/GenericDev (IEC)

#### GenericDevice.st
```iecst
FUNCTION_BLOCK GenericDevice

	(* CLOCK HANDLER *)
	IF (DeviceClock AND (DeviceTimer > 0))THEN
		DeviceTimer := DeviceTimer - 1;
	END_IF;

	(* DEVICE SENSORS HANDLER *)
	CASE (DeviceType AND DEVICE_FEEDBACK_MASK) OF

		DEVICE_WITH_ENABLE_FEEDBACK:

			DeviceDisabledSensor := NOT DeviceEnabledSensor AND
			((DeviceState = DeviceDisabledState) OR (DeviceState = DeviceDisablePhaseState AND DeviceTimeout));

			DeviceDisabled 		 := NOT DeviceEnabled AND
			((DeviceState = DeviceDisabledState) OR (DeviceState = DeviceDisablePhaseState AND DeviceTimeout));

		DEVICE_WITH_DISABLE_FEEDBACK :

			DeviceEnabled 		:= NOT DeviceDisabled AND
			((DeviceState = DeviceEnabledState) OR (DeviceState = DeviceEnablePhaseState AND DeviceTimeout));

			DeviceEnabledSensor := NOT DeviceDisabledSensor AND
			((DeviceState = DeviceEnabledState) OR (DeviceState = DeviceEnablePhaseState AND DeviceTimeout));

		DEVICE_WITHOUT_FEEDBACK:

			DeviceEnabled  		 := (DeviceState = DeviceEnabledState) OR (DeviceState = DeviceEnablePhaseState AND DeviceTimeout);

			DeviceDisabled 		 := (DeviceState = DeviceDisabledState) OR (DeviceState = DeviceDisablePhaseState AND DeviceTimeout);

			DeviceEnabledSensor  := (DeviceState = DeviceEnabledState) OR ((DeviceState = DeviceEnablePhaseState) AND DeviceTimeout);

			DeviceDisabledSensor := (DeviceState = DeviceDisabledState) OR ((DeviceState = DeviceDisablePhaseState) AND DeviceTimeout);

	END_CASE;

	(* INITIALIZATION HANDLER *)
	IF (DeviceOperation = INIT) THEN

		CASE (DeviceType AND DEVICE_FEEDBACK_MASK) OF

			DEVICE_WITH_ENABLE_FEEDBACK:

				DeviceDisabled := NOT DeviceEnabled;

			DEVICE_WITH_DISABLE_FEEDBACK:

				DeviceEnabled := NOT DeviceDisabled;

			DEVICE_WITHOUT_FEEDBACK:

				DeviceEnabled  := DeviceEnablePreset;
				DeviceDisabled := NOT DeviceEnabled;

		END_CASE;

		DeviceEnableRequest  := FALSE;
		DeviceDisableRequest := FALSE;

		IF (DeviceEnablePreset) THEN
			EnableDevice := TRUE;
			DeviceTimer  := DeviceEnableTime;

			IF (NOT (DeviceDisabled AND DeviceEnabled)) THEN
				DeviceState := DeviceEnablePhaseState;
			ELSE
				DeviceState := DeviceEnabledState;
			END_IF;

			DeviceNotInitialized := NOT DeviceEnabled OR DeviceDisabled;

		ELSE
			EnableDevice := FALSE;
			DeviceTimer := DeviceDisableTime;

			IF (NOT (DeviceDisabled AND DeviceEnabled)) THEN
				DeviceState := DeviceDisablePhaseState;
			ELSE
				DeviceState := DeviceDisabledState;
			END_IF;

			DeviceNotInitialized := (DeviceEnabled OR NOT DeviceDisabled);
		END_IF;

	END_IF;

	(* DEVICE CONTROL HANDLER *)
	CASE (DeviceState) OF

		DeviceDisabledState:

			DeviceDisableRequest := FALSE;
			IF (DeviceEnableRequest) THEN
				EnableDevice := TRUE;
				DeviceTimer  := DeviceEnableTime;
				DeviceState  := DeviceEnablePhaseState;
			END_IF;

		DeviceEnablePhaseState:

			IF DeviceDisableRequest THEN
				DeviceEnableRequest	:= FALSE;
				EnableDevice	    := FALSE;
				DeviceTimer	        := DeviceDisableTime;
				DeviceState	        := DeviceDisablePhaseState;
			END_IF;

			IF DeviceEnabledSensor THEN
				DeviceEnableRequest := FALSE;
				DeviceTimer	        := 0;
				DeviceState         := DeviceEnabledState;
			END_IF;

		DeviceEnabledState:

			DeviceEnableRequest	:= FALSE;
			IF DeviceDisableRequest THEN
				EnableDevice := FALSE;
				DeviceTimer	 := DeviceDisableTime;
				DeviceState  := DeviceDisablePhaseState;
			END_IF;

		DeviceDisablePhaseState:

			IF DeviceEnableRequest THEN
				DeviceDisableRequest := FALSE;
				EnableDevice		 := TRUE;
				DeviceTimer			 := DeviceEnableTime;
				DeviceState			 := DeviceEnablePhaseState;
			END_IF;

			IF DeviceDisabledSensor THEN
				DeviceDisableRequest := FALSE;
				DeviceTimer          := 0;
				DeviceState 		 := DeviceDisabledState;
			END_IF;

	END_CASE;

	(* DEVICE DIAGNOSIS HANDLER *)
	DeviceTimeout 			  := (DeviceTimer = 0);

	DeviceDisabledSensorFault := ((NOT EnableDevice AND NOT DeviceDisabledSensor AND NOT DeviceEnabledSensor) OR
	(EnableDevice AND DeviceDisabledSensor AND DeviceEnabledSensor)) AND DeviceTimeout;

	DeviceEnabledSensorFault  := ((NOT EnableDevice AND DeviceDisabledSensor AND DeviceEnabledSensor) OR
	(EnableDevice AND NOT DeviceDisabledSensor AND NOT DeviceEnabledSensor)) AND DeviceTimeout;

	DeviceActuatorFault 	  := ((NOT EnableDevice AND NOT DeviceDisabledSensor AND DeviceEnabledSensor) OR
	(EnableDevice AND DeviceDisabledSensor AND NOT DeviceEnabledSensor)) AND DeviceTimeout;

	DeviceFault 			  := DeviceDisabledSensorFault OR DeviceEnabledSensorFault OR DeviceActuatorFault;

	(* DEVICE ACTUATORS HANDLER *)
	CASE (DeviceType AND DEVICE_ACTUATION_MASK) OF

		DEVICE_WITH_DOUBLE_ACTUATION:

			DisableDevice := NOT EnableDevice;

		DEVICE_WITH_DA_NO_RETAIN:

			EnableDevice  := EnableDevice AND (DeviceState = DeviceEnablePhaseState);
			DisableDevice := NOT EnableDevice AND (DeviceState = DeviceDisablePhaseState);

	END_CASE;

END_FUNCTION_BLOCK
```

#### Types.typ - Exported data types
```iecst
TYPE
	DeviceStateType :
		(
		DeviceDisabledState,
		DeviceEnablePhaseState,
		DeviceEnabledState,
		DeviceDisablePhaseState
		);
END_TYPE
```

#### Constants.var - Exported constants
```iecst
VAR CONSTANT
	DEVICE_WITHOUT_FEEDBACK : INT := 2#01000000;
	DEVICE_WITH_ENABLE_FEEDBACK : INT := 2#00010000;
	DEVICE_WITH_DISABLE_FEEDBACK : INT := 2#00100000;
	DEVICE_WITH_DOUBLE_FEEDBACK : INT := 2#00110000;
	DEVICE_WITH_SINGLE_ACTUATION : INT := 2#00000001;
	DEVICE_WITH_DOUBLE_ACTUATION : INT := 2#00000011;
	DEVICE_WITH_DA_NO_RETAIN : INT := 2#00000010;
	DEVICE_FEEDBACK_MASK : INT := 2#11110000;
	DEVICE_ACTUATION_MASK : INT := 2#00001111;
	END_VAR
```

#### GenericDev.fun - Exported functions and function blocks
```iecst
{REDUND_ERROR} {REDUND_UNREPLICABLE} FUNCTION_BLOCK GenericDevice (*TODO: Add your comment here*) (*$GROUP=User,$CAT=User,$GROUPICON=User.png,$CATICON=User.png*)
	VAR_INPUT
		DeviceOperation : {REDUND_UNREPLICABLE} INT;
		DeviceType : {REDUND_UNREPLICABLE} INT;
		DeviceEnabledSensor : {REDUND_UNREPLICABLE} BOOL;
		DeviceDisabledSensor : {REDUND_UNREPLICABLE} BOOL;
		DeviceClock : {REDUND_UNREPLICABLE} BOOL;
		DeviceEnableTime : {REDUND_UNREPLICABLE} INT;
		DeviceDisableTime : {REDUND_UNREPLICABLE} INT;
		DeviceDiagnosticsEnabled : {REDUND_UNREPLICABLE} BOOL;
		DeviceEnablePreset : {REDUND_UNREPLICABLE} BOOL;
		DeviceEnabled : {REDUND_UNREPLICABLE} BOOL;
		DeviceDisabled : {REDUND_UNREPLICABLE} BOOL;
	END_VAR
	VAR_OUTPUT
		EnableDevice : {REDUND_UNREPLICABLE} BOOL;
		DisableDevice : {REDUND_UNREPLICABLE} BOOL;
		DeviceEnabledSensorFault : {REDUND_UNREPLICABLE} BOOL;
		DeviceDisabledSensorFault : {REDUND_UNREPLICABLE} BOOL;
		DeviceActuatorFault : {REDUND_UNREPLICABLE} BOOL;
		DeviceFault : {REDUND_UNREPLICABLE} BOOL;
		DeviceNotInitialized : {REDUND_UNREPLICABLE} BOOL;
	END_VAR
	VAR_IN_OUT
		DeviceEnableRequest : BOOL;
		DeviceDisableRequest : BOOL;
	END_VAR
	VAR
		DeviceState : {REDUND_UNREPLICABLE} DeviceStateType;
		DeviceTimer : {REDUND_UNREPLICABLE} INT;
		DeviceTimeout : {REDUND_UNREPLICABLE} BOOL;
	END_VAR
	VAR CONSTANT
		INIT : INT := 0;
		RUN : INT := 1;
	END_VAR
END_FUNCTION_BLOCK
```

### Library Logical/Libraries/GenericAx (IEC)

#### GenericAxis.st
```iecst
(* TODO: Add your comment here *)
FUNCTION_BLOCK GenericAxis

	CASE (AxisState) OF

		CheckCommand:

			IF Command = IDLE THEN
				InPosition	:= FALSE;
				InVelocity	:= FALSE;
				Timer		:= DeviceTimer;
				DeviceFault	:= FALSE;
			END_IF;

			IF Command = CHANGE_POSITION THEN
				TargetPosition	:= NewSetPoint;
				AxisState		:= WaitTargetPosition;
			END_IF;

			IF Command = CHANGE_VELOCITY THEN
				TargetVelocity := NewSetPoint;
				AxisState	   := WaitTargetVelocity;
			END_IF;

			IF Command = EMERGENCY_STOP_REQUEST THEN
				TargetPosition	:= ActualPosition;
				TargetVelocity	:= 0;
				IF (ActualPosition = TargetPosition AND ActualVelocity = TargetVelocity) THEN
					InPosition	:= TRUE;
					InVelocity	:= TRUE;
					AxisState	:= CheckCommand;
				END_IF;
			END_IF;

		WaitTargetPosition:

			IF (ActualPosition = NewSetPoint AND TGT_SENSOR) THEN
				InPosition	:= TRUE;
				AxisState	:= CheckCommand;
			END_IF;

			Timer := Timer	- 1;
			IF Timer = 0 THEN
				DeviceFault	:= TRUE;
				AxisState	:= FaultState;
			END_IF;

		WaitTargetVelocity:

			IF ActualVelocity = NewSetPoint THEN
				InVelocity	:= TRUE;
				AxisState	:= CheckCommand;
			END_IF;

			Timer := Timer	- 1;
			IF Timer = 0 THEN
				DeviceFault	:= TRUE;
				AxisState	:= FaultState;
			END_IF;

		FaultState:

			IF Reset THEN
				DeviceFault	:= FALSE;
				AxisState	:= CheckCommand;
			END_IF;

	END_CASE;

END_FUNCTION_BLOCK
```

#### Types.typ - Exported data types
```iecst
TYPE
	GA_State :
		(
		CheckCommand,
		WaitTargetPosition,
		WaitTargetVelocity,
		FaultState
		);
END_TYPE
```

#### Constants.var - Exported constants
```iecst
VAR CONSTANT
	IDLE : WORD := 0;
	CHANGE_VELOCITY : WORD := 1;
	CHANGE_POSITION : WORD := 2;
	EMERGENCY_STOP_REQUEST : WORD := 3;
END_VAR
```

#### GenericAx.fun - Exported functions and function blocks
```iecst
FUNCTION_BLOCK GenericAxis
	VAR_INPUT
		Command : WORD := 95;
		ActualPosition : REAL;
		ActualVelocity : REAL;
		NewSetPoint : REAL;
		DeviceTimer : INT;
		TGT_SENSOR : BOOL;
	END_VAR
	VAR_OUTPUT
		TargetVelocity : REAL;
		TargetPosition : REAL;
		InPosition : BOOL;
		InVelocity : BOOL;
		DeviceFault : BOOL;
	END_VAR
	VAR
		AxisState : GA_State := CheckCommand;
		Timer : INT;
	END_VAR
	VAR_INPUT
		Reset : BOOL;
	END_VAR
END_FUNCTION_BLOCK
```

### Library Logical/Libraries/SignalMng (IEC)

#### SignalManager.st
```iecst
FUNCTION_BLOCK SignalManager

	CASE OperationType OF

(* 0 *)	START_CONFIGURATION: (* Reset signals counts *)

			NumberOfAlarms 	    := 0;
			NumberOfAnomalies   := 0;
			NumberOfWarnings 	:= 0;
			NumberOfInformation := 0;

(* 1 *)	CONFIGURATION: (* counting signals *)

			CASE (SignalType AND SIGNAL_TYPE_MASK) OF
				ALARM:
					NumberOfAlarms 	    := NumberOfAlarms + 1;

				ANOMALY:
					NumberOfAnomalies   := NumberOfAnomalies + 1;

				WARNING:
					NumberOfWarnings    := NumberOfWarnings + 1;

				INFORMATION:
					NumberOfInformation := NumberOfInformation + 1;
			END_CASE

(* 2 *)	START_GENERATION:

			AuxResetEnable	   := FALSE;
			ResetEnable 	   := FALSE;
			SignalOutputs 	   := NONE;
			ResetActivation    := Reset AND NOT ResetOld;
			ResetOld 		   := Reset;
			AuxResetActivation := KeyReset AND NOT KeyResetOld;
			KeyResetOld		   := KeyReset;

(* 3 *)	GENERATION:

			CASE (SignalType AND SIGNAL_TYPE_MASK) OF
				ALARM:
					Index 	  := NumberOfActiveAlarms;
					BaseIndex := 0;
					Condition := TRUE;

				ANOMALY:
					Index 	  := NumberOfActiveAnomalies;
					BaseIndex := NumberOfAlarms;
					Condition := TRUE;

				WARNING:
					Index 	  := NumberOfActiveWarning;
					BaseIndex := NumberOfAlarms + NumberOfAnomalies;
					Condition := FALSE;

				INFORMATION:
					Index 	  := NumberOfActiveInformation;
					BaseIndex := NumberOfAlarms + NumberOfAnomalies + NumberOfWarnings;
					Condition := FALSE;
			END_CASE

			IF ActivationSignal AND NOT Signals[SignalCode] THEN
				Signals[SignalCode] 				 := TRUE;
				Index 								 := Index + 1;
				ActiveSignalCodes[BaseIndex + Index] := SignalCode;
			END_IF

			AuxResetRequired := ((SignalType AND AUX_RESET) = AUX_RESET);

			IF (Condition AND Signals[SignalCode] AND NOT ActivationSignal AND (ActiveSignalCodes[BaseIndex + 1] = SignalCode) AND AuxResetRequired) THEN
				AuxResetEnable := TRUE;
			END_IF

			IF (Condition AND Signals[SignalCode] AND NOT ActivationSignal AND (ActiveSignalCodes[BaseIndex + 1] = SignalCode) AND NOT AuxResetRequired) THEN
				ResetEnable := TRUE;
//				AuxResetEnable := TRUE;
			END_IF

			IF ((ResetActivation OR NOT Condition) AND Signals[SignalCode] AND NOT ActivationSignal AND (ActiveSignalCodes[BaseIndex + 1] = SignalCode) AND NOT AuxResetRequired) THEN
				Signals[SignalCode] := FALSE;

				FOR i := 2 TO Index DO
					ActiveSignalCodes[BaseIndex + i-1] := ActiveSignalCodes[BaseIndex + i];
				END_FOR;

				ActiveSignalCodes[BaseIndex + Index] := 0;
				Index 								 := Index - 1;
				ResetActivation 					 := FALSE;
			END_IF

			IF ((AuxResetActivation OR NOT Condition) AND Signals[SignalCode] AND NOT ActivationSignal AND (ActiveSignalCodes[BaseIndex + 1] = SignalCode) (*AND AuxResetRequired*)) THEN
				Signals[SignalCode] := FALSE;

				FOR i := 2 TO Index DO
					ActiveSignalCodes[BaseIndex + i-1] := ActiveSignalCodes[BaseIndex + i];
				END_FOR;

				ActiveSignalCodes[BaseIndex + Index] := 0;
				Index 								 := Index - 1;
				AuxResetActivation 					 := FALSE;
			END_IF

			CASE (SignalType AND SIGNAL_TYPE_MASK) OF
				ALARM:
					NumberOfActiveAlarms := Index;

				ANOMALY:
					NumberOfActiveAnomalies := Index;

				WARNING:
					NumberOfActiveWarning := Index;

				INFORMATION:
					NumberOfActiveInformation := Index;
			END_CASE

			IF Signals[SignalCode] THEN
				SignalOutputs := SignalOutputs OR SignalOutput;
			END_IF

(* 4 *)	RUN:

			FirstActiveSignalIndex	:= ActiveSignalCodes[1];
			SecondActiveSignalIndex	:= ActiveSignalCodes[2];
			ThirdActiveSignalIndex	:= ActiveSignalCodes[3];
			FourthActiveSignalIndex	:= ActiveSignalCodes[4];
			FifthActiveSignalIndex  := ActiveSignalCodes[5];

			LastInformationIndex 	:= NumberOfAlarms + NumberOfAnomalies + NumberOfWarnings + NumberOfActiveInformation;

			IF NumberOfActiveInformation > 0 THEN
				SignalTypeInformation	:= TRUE;
			ELSE
				SignalTypeInformation	:= FALSE;
			END_IF

			LastAnomalyIndex := NumberOfAlarms + NumberOfAnomalies + NumberOfActiveAnomalies;

			IF NumberOfActiveAnomalies > 0 THEN
				SignalTypeAnomaly	:= TRUE;
			ELSE
				SignalTypeAnomaly	:= FALSE;
			END_IF

			LastWarningIndex := NumberOfAlarms + NumberOfActiveWarning;

			IF NumberOfActiveWarning > 0 THEN
				SignalTypeWarning	:= TRUE;
			ELSE
				SignalTypeWarning	:= FALSE;
			END_IF

			IF NumberOfActiveAlarms = 2 AND ResetEnable AND AuxResetEnable THEN
				NumberOfActiveAlarms := 1;
			END_IF

			IF NumberOfActiveAlarms > 0 THEN
				SignalTypeAlarm	:= TRUE;
			ELSE
				SignalTypeAlarm	:= FALSE;
			END_IF

	END_CASE

// Output of the alarm registry log

//	First alarm
	IF 	FirstActiveSignalIndex = 1	THEN
		Firstslot:= 'Turnpusher BROKEN';
	ELSIF FirstActiveSignalIndex = 2 THEN
		Firstslot:= 'Pusher BROKEN';
	ELSIF FirstActiveSignalIndex = 3 THEN
		Firstslot:= 'Crane Pusher X-axis BROKEN';
	ELSIF FirstActiveSignalIndex = 4 THEN
		Firstslot:= 'Crane Pusher Z-axis BROKEN';
	ELSIF FirstActiveSignalIndex = 5 THEN
		Firstslot:= 'Vacuum BROKEN';
	ELSIF FirstActiveSignalIndex = 6 THEN
		Firstslot:= 'Pallet Fork BROKEN';
	ELSIF FirstActiveSignalIndex = 7 THEN
		Firstslot:= 'Pallets OVER';
	ELSIF FirstActiveSignalIndex = 8 THEN
		Firstslot:= 'Carriage BROKEN';
	ELSIF FirstActiveSignalIndex = 9 THEN
		Firstslot:= 'Gantry Crane BROKEN';
	ELSIF FirstActiveSignalIndex = 10 THEN
		Firstslot:= 'Box Crane BROKEN';
	ELSIF FirstActiveSignalIndex = 11 THEN
		Firstslot:= 'Pallet Lifter BROKEN';
	ELSIF FirstActiveSignalIndex = 12 THEN
			Firstslot:= 'Pallets ALMOST OVER';
	ELSIF FirstActiveSignalIndex = 13 THEN
		Firstslot:= 'On Phase Stop REQUESTED';
	ELSIF FirstActiveSignalIndex = 14 THEN
		Firstslot:= 'Emergency Stop REQUESTED';
	ELSIF FirstActiveSignalIndex = 15 THEN
		Firstslot:= 'Cartboards ALMOST OVER';
	ELSIF FirstActiveSignalIndex = 16 THEN
		Firstslot:= 'Cartboards OVER';
	ELSIF FirstActiveSignalIndex = 17 THEN
		Firstslot:= 'Conveyor 1 BROKEN';
	ELSIF FirstActiveSignalIndex = 18 THEN
		Firstslot:= 'Conveyor 2 BROKEN';
	ELSIF FirstActiveSignalIndex = 19 THEN
		Firstslot:= 'Conveyor 3 BROKEN';
//	ELSIF FirstActiveSignalIndex = 20 THEN
//		Firstslot:= 'Cartboards FAULT';
	ELSIF FirstActiveSignalIndex = 21 THEN
		Firstslot:= 'Slide Rail BROKEN';
	ELSIF FirstActiveSignalIndex = 22 THEN
		Firstslot:= 'Pallet Conveyor 1 BROKEN';
	ELSIF FirstActiveSignalIndex = 23 THEN
		Firstslot:= 'Pallet Conveyor 2 BROKEN';
	ELSE
		Firstslot:= '-';
	END_IF;

//	Second alarm
	IF 	SecondActiveSignalIndex = 1	THEN
		Secondslot := 'Turnpusher BROKEN';
	ELSIF SecondActiveSignalIndex = 2 THEN
		Secondslot:= 'Pusher BROKEN';
	ELSIF SecondActiveSignalIndex = 3 THEN
		Secondslot:= 'Crane Pusher X-axis BROKEN';
	ELSIF SecondActiveSignalIndex = 4 THEN
		Secondslot:= 'Crane Pusher Z-axis BROKEN';
	ELSIF SecondActiveSignalIndex = 5 THEN
		Secondslot:= 'Vacuum BROKEN';
	ELSIF SecondActiveSignalIndex = 6 THEN
		Secondslot:= 'Pallet Fork BROKEN';
	ELSIF SecondActiveSignalIndex = 7 THEN
		Secondslot:= 'Pallets OVER';
	ELSIF SecondActiveSignalIndex = 8 THEN
		Secondslot:= 'Carriage BROKEN';
	ELSIF SecondActiveSignalIndex = 9 THEN
		Secondslot:= 'Gantry Crane BROKEN';
	ELSIF SecondActiveSignalIndex = 10 THEN
		Secondslot:= 'Box Crane BROKEN';
	ELSIF SecondActiveSignalIndex = 11 THEN
		Secondslot:= 'Pallet Lifter BROKEN';
	ELSIF SecondActiveSignalIndex = 12 THEN
		Secondslot:= 'Pallets ALMOST OVER';
	ELSIF SecondActiveSignalIndex = 13 THEN
		Secondslot:= 'On Phase Stop REQUESTED';
	ELSIF SecondActiveSignalIndex = 14 THEN
		Secondslot:= 'Emergency Stop REQUESTED';
	ELSIF SecondActiveSignalIndex = 15 THEN
 		Secondslot:= 'Cartboards ALMOST OVER';
	ELSIF SecondActiveSignalIndex = 16 THEN
		Secondslot:= 'Cartboards OVER';
	ELSIF SecondActiveSignalIndex = 17 THEN
		Secondslot:= 'Conveyor 1 BROKEN';
	ELSIF SecondActiveSignalIndex = 18 THEN
		Secondslot:= 'Conveyor 2 BROKEN';
	ELSIF SecondActiveSignalIndex = 19 THEN
		Secondslot:= 'Conveyor 3 BROKEN';
//	ELSIF SecondActiveSignalIndex = 20 THEN
//		Secondslot:= 'Cartboard FAULT';
	ELSIF SecondActiveSignalIndex = 21 THEN
		Secondslot:= 'Slide Rail BROKEN';
	ELSIF SecondActiveSignalIndex = 22 THEN
		Secondslot:= 'Pallet Conveyor 1 BROKEN';
	ELSIF SecondActiveSignalIndex = 23 THEN
		Secondslot:= 'Pallet Conveyor 2 BROKEN';
	ELSE
		Secondslot:= '-';
	END_IF;

// 	Third alarm
	IF 	ThirdActiveSignalIndex = 1	THEN
		Thirdslot:= 'Turnpusher BROKEN';
	ELSIF ThirdActiveSignalIndex = 2 THEN
		Thirdslot:= 'Pusher BROKEN';
	ELSIF ThirdActiveSignalIndex = 3 THEN
		Thirdslot:= 'Crane Pusher X-axis BROKEN';
	ELSIF ThirdActiveSignalIndex = 4 THEN
		Thirdslot:= 'Crane Pusher Z-axis BROKEN';
	ELSIF ThirdActiveSignalIndex = 5 THEN
		Thirdslot:= 'Vacuum BROKEN';
	ELSIF ThirdActiveSignalIndex = 6 THEN
		Thirdslot:= 'Pallet Fork BROKEN';
	ELSIF ThirdActiveSignalIndex = 7 THEN
		Thirdslot:= 'Pallets OVER';
	ELSIF ThirdActiveSignalIndex = 8 THEN
		Thirdslot:= 'Carriage BROKEN';
	ELSIF ThirdActiveSignalIndex = 9 THEN
		Thirdslot:= 'Gantry Crane BROKEN';
	ELSIF ThirdActiveSignalIndex = 10 THEN
		Thirdslot:= 'Box Crane BROKEN';
	ELSIF ThirdActiveSignalIndex = 11 THEN
		Thirdslot:= 'Pallet Lifter BROKEN';
	ELSIF ThirdActiveSignalIndex = 12 THEN
		Thirdslot:= 'Pallets ALMOST OVER';
	ELSIF ThirdActiveSignalIndex = 13 THEN
		Thirdslot:= 'On Phase Stop REQUESTED';
	ELSIF ThirdActiveSignalIndex = 14 THEN
		Thirdslot:= 'Emergency Stop REQUESTED';
	ELSIF ThirdActiveSignalIndex = 15 THEN
		Thirdslot:= 'Cartboards ALMOST OVER';
	ELSIF ThirdActiveSignalIndex = 16 THEN
		Thirdslot:= 'Cartboards OVER';
	ELSIF ThirdActiveSignalIndex = 17 THEN
		Thirdslot:= 'Conveyor 1 BROKEN';
	ELSIF ThirdActiveSignalIndex = 18 THEN
		Thirdslot:= 'Conveyor 2 BROKEN';
	ELSIF ThirdActiveSignalIndex = 19 THEN
		Thirdslot:= 'Conveyor 3 BROKEN';
//	ELSIF ThirdActiveSignalIndex = 20 THEN
//		Thirdslot:= 'Cartboards FAULT';
	ELSIF ThirdActiveSignalIndex = 21 THEN
		Thirdslot:= 'Slide Rail BROKEN';
	ELSIF ThirdActiveSignalIndex = 22 THEN
		Thirdslot:= 'Pallet Conveyor 1 BROKEN';
	ELSIF ThirdActiveSignalIndex = 23 THEN
		Thirdslot:= 'Pallet Conveyor 2 BROKEN';
	ELSE
		Thirdslot:= '-';
	END_IF

//	Fourth alarm
	IF 	FourthActiveSignalIndex = 1	THEN
		Fourthslot:= 'Turnpusher BROKEN';
	ELSIF FourthActiveSignalIndex = 2 THEN
		Fourthslot:= 'Pusher BROKEN';
	ELSIF FourthActiveSignalIndex = 3 THEN
		Fourthslot:= 'Crane Pusher X-axis BROKEN';
	ELSIF FourthActiveSignalIndex = 4 THEN
		Fourthslot:= 'Crane Pusher Z-axis BROKEN';
	ELSIF FourthActiveSignalIndex = 5 THEN
		Fourthslot:= 'Vacuum BROKEN';
	ELSIF FourthActiveSignalIndex = 6 THEN
		Fourthslot:= 'Pallet Fork BROKEN';
	ELSIF FourthActiveSignalIndex = 7 THEN
		Fourthslot:= 'Pallets OVER';
	ELSIF FourthActiveSignalIndex = 8 THEN
		Fourthslot:= 'Carriage BROKEN';
	ELSIF FourthActiveSignalIndex = 9 THEN
		Fourthslot:= 'Gantry Crane BROKEN';
	ELSIF FourthActiveSignalIndex = 10 THEN
		Fourthslot:= 'Box Crane BROKEN';
	ELSIF FourthActiveSignalIndex = 11 THEN
		Fourthslot:= 'Pallet Lifter BROKEN';
	ELSIF FourthActiveSignalIndex = 12 THEN
		Fourthslot:= 'Pallets ALMOST OVER';
	ELSIF FourthActiveSignalIndex = 13 THEN
		Fourthslot:= 'On Phase Stop REQUESTED';
	ELSIF FourthActiveSignalIndex = 14 THEN
		Fourthslot:= 'Emergency Stop REQUESTED';
	ELSIF FourthActiveSignalIndex = 15 THEN
		Fourthslot:= 'Cartboards ALMOST OVER';
	ELSIF FourthActiveSignalIndex = 16 THEN
		Fourthslot:= 'Cartboards OVER';
	ELSIF FourthActiveSignalIndex = 17 THEN
		Fourthslot:= 'Conveyor 1 BROKEN';
	ELSIF FourthActiveSignalIndex = 18 THEN
		Fourthslot:= 'Conveyor 2 BROKEN';
	ELSIF FourthActiveSignalIndex = 19 THEN
		Fourthslot:= 'Conveyor 3 BROKEN';
//	ELSIF FourthActiveSignalIndex = 20 THEN
//		Fourthslot:= 'Cartboards FAULT';
	ELSIF FourthActiveSignalIndex = 21 THEN
		Fourthslot:= 'Slide Rail BROKEN';
	ELSIF FourthActiveSignalIndex = 22 THEN
		Fourthslot:= 'Pallet Conveyor 1 BROKEN';
	ELSIF FourthActiveSignalIndex = 23 THEN
		Fourthslot:= 'Pallet Conveyor 2 BROKEN';
	ELSE
		Fourthslot:= '-';
	END_IF

	//	Fifth alarm
	IF 	FifthActiveSignalIndex = 1	THEN
		Fifthslot:= 'Turnpusher BROKEN';
	ELSIF FifthActiveSignalIndex = 2 THEN
		Fifthslot:= 'Pusher BROKEN';
	ELSIF FifthActiveSignalIndex = 3 THEN
		Fifthslot:= 'Crane Pusher X-axis BROKEN';
	ELSIF FifthActiveSignalIndex = 4 THEN
		Fifthslot:= 'Crane Pusher Z-axis BROKEN';
	ELSIF FifthActiveSignalIndex = 5 THEN
		Fifthslot:= 'Vacuum BROKEN';
	ELSIF FifthActiveSignalIndex = 6 THEN
		Fifthslot:= 'Pallet Fork BROKEN';
	ELSIF FifthActiveSignalIndex = 7 THEN
		Fifthslot:= 'Pallets OVER';
	ELSIF FifthActiveSignalIndex = 8 THEN
		Fifthslot:= 'Carriage BROKEN';
	ELSIF FifthActiveSignalIndex = 9 THEN
		Fifthslot:= 'Gantry Crane BROKEN';
	ELSIF FifthActiveSignalIndex = 10 THEN
		Fifthslot:= 'Box Crane BROKEN';
	ELSIF FifthActiveSignalIndex = 11 THEN
		Fifthslot:= 'Pallet Lifter BROKEN';
	ELSIF FifthActiveSignalIndex = 12 THEN
		Fifthslot:= 'Pallets ALMOST OVER';
	ELSIF FifthActiveSignalIndex = 13 THEN
		Fifthslot:= 'On Phase Stop REQUESTED';
	ELSIF FifthActiveSignalIndex = 14 THEN
		Fifthslot:= 'Emergency Stop REQUESTED';
	ELSIF FifthActiveSignalIndex = 15 THEN
		Fifthslot:= 'Cartboards ALMOST OVER';
	ELSIF FifthActiveSignalIndex = 16 THEN
		Fifthslot:= 'Cartboards OVER';
	ELSIF FifthActiveSignalIndex = 17 THEN
		Fifthslot:= 'Conveyor 1 BROKEN';
	ELSIF FifthActiveSignalIndex = 18 THEN
		Fifthslot:= 'Conveyor 2 BROKEN';
	ELSIF FifthActiveSignalIndex = 19 THEN
		Fifthslot:= 'Conveyor 3 BROKEN';
//	ELSIF FifthActiveSignalIndex = 20 THEN
//		Fifthslot:= 'Cartboards FAULT';
	ELSIF FifthActiveSignalIndex = 21 THEN
		Fifthslot:= 'Slide Rail BROKEN';
	ELSIF FifthActiveSignalIndex = 22 THEN
		Fifthslot:= 'Pallet Conveyor 1 BROKEN';
	ELSIF FifthActiveSignalIndex = 23 THEN
		Fifthslot:= 'Pallet Conveyor 2 BROKEN';
	ELSE
		Fifthslot:= '-';
	END_IF

END_FUNCTION_BLOCK
```

#### Constants.var - Exported constants
```iecst
VAR CONSTANT
	INIT : INT := 0;
	RUN : INT := 1;
	START_CONFIGURATION : INT := 2;
	CONFIGURATION : INT := 3;
	START_GENERATION : INT := 4;
	GENERATION : INT := 5;
	ALARM : DINT := 2#0000000000000001;
	ANOMALY : DINT := 2#0000000000000010;
	WARNING : DINT := 2#0000000000000011;
	INFORMATION : DINT := 2#0000000000000100;
	AUX_RESET : DINT := 2#0000001000000000;
	UNCONDITIONED_RESET : DINT := 2#0100000000000000;
	AUTO_CONDITIONED_RESET : DINT := 2#0010000000000000;
	AUTO_PROVISIONAL_RESET : DINT := 2#0001000000000000;
	AUTO_PRIORITY_RESET : DINT := 2#0000100000000000;
	AUTO_RESET : DINT := 2#0000010000000000;
	SIGNAL_TYPE_MASK : DINT := 2#0000000000000111;
	NONE : DWORD := 16#0000;
	EMERGENCY_STOP : DWORD := 16#0001;
	IMMEDIATE_STOP : DWORD := 16#0002;
	ON_PHASE_STOP : DWORD := 16#0004;
	MACHINE_OUT_OF_PHASE : DWORD := 16#0100;
	MACHINE_INHIBITION : DWORD := 16#0200;
	MATERIALS_RUN_OUT_LAMP : DWORD := 16#0400;
	MATERIALS_RUN_OUT_BUZZER : DWORD := 16#0800;
	IO_DIAGNOSTIC_INHIBITION : DWORD := 16#8000;
END_VAR
```

#### SignalMng.fun - Exported functions and function blocks
```iecst
{REDUND_ERROR} FUNCTION_BLOCK SignalManager (*TODO: Add your comment here*) (*$GROUP=User,$CAT=User,$GROUPICON=User.png,$CATICON=User.png*)
	VAR_INPUT
		OperationType : {REDUND_UNREPLICABLE} INT;
		SignalType : {REDUND_UNREPLICABLE} DINT := 0;
		SignalCode : {REDUND_UNREPLICABLE} INT := 0;
		SignalOutput : {REDUND_UNREPLICABLE} DWORD := 0;
		ActivationSignal : {REDUND_UNREPLICABLE} BOOL := FALSE;
		AutoResetSignal : {REDUND_UNREPLICABLE} BOOL := FALSE;
		Reset : {REDUND_UNREPLICABLE} BOOL;
		KeyReset : {REDUND_UNREPLICABLE} BOOL;
	END_VAR
	VAR_OUTPUT
		SignalOutputs : {REDUND_UNREPLICABLE} DWORD;
		SignalPriorityCode : {REDUND_UNREPLICABLE} WORD;
		ResetEnable : {REDUND_UNREPLICABLE} BOOL;
		AuxResetEnable : {REDUND_UNREPLICABLE} BOOL;
		SignalTypeAlarm : {REDUND_UNREPLICABLE} BOOL;
		SignalTypeAnomaly : {REDUND_UNREPLICABLE} BOOL;
		SignalTypeWarning : {REDUND_UNREPLICABLE} BOOL;
		SignalTypeInformation : {REDUND_UNREPLICABLE} BOOL;
		NumberOfAlarms : {REDUND_UNREPLICABLE} INT;
		NumberOfAnomalies : {REDUND_UNREPLICABLE} INT;
		NumberOfWarnings : {REDUND_UNREPLICABLE} INT;
		NumberOfInformation : {REDUND_UNREPLICABLE} INT;
		ActiveSignalCodes : {REDUND_UNREPLICABLE} ARRAY[1..20] OF INT;
		NumberOfActiveAlarms : {REDUND_UNREPLICABLE} INT := 0;
		NumberOfActiveAnomalies : {REDUND_UNREPLICABLE} INT := 0;
		NumberOfActiveWarning : {REDUND_UNREPLICABLE} INT := 0;
		NumberOfActiveInformation : {REDUND_UNREPLICABLE} INT := 0;
		SignalManagementError : {REDUND_UNREPLICABLE} BOOL;
		FirstSignalIndex : INT;
		FirstActiveSignalIndex : INT;
		SecondActiveSignalIndex : INT;
		ThirdActiveSignalIndex : INT;
		FourthActiveSignalIndex : INT;
		FifthActiveSignalIndex : INT;
	END_VAR
	VAR
		ResetSignalsEnable : {REDUND_UNREPLICABLE} BOOL;
		AuxResetActivation : {REDUND_UNREPLICABLE} BOOL;
		ResetActivation : {REDUND_UNREPLICABLE} BOOL;
		SignalRequest : {REDUND_UNREPLICABLE} BOOL;
		SignalAckRequest : {REDUND_UNREPLICABLE} BOOL;
		Signals : {REDUND_UNREPLICABLE} ARRAY[1..23] OF BOOL;
		LastSignalIndex : {REDUND_UNREPLICABLE} INT;
		ActiveSignalRequest : {REDUND_UNREPLICABLE} BOOL;
		ActiveSignalRequestAck : {REDUND_UNREPLICABLE} BOOL;
		LastActiveSignalIndex : {REDUND_UNREPLICABLE} INT;
		ResetOld : {REDUND_UNREPLICABLE} BOOL;
		KeyResetOld : {REDUND_UNREPLICABLE} BOOL;
		Index : {REDUND_UNREPLICABLE} INT;
		BaseIndex : {REDUND_UNREPLICABLE} INT;
		Condition : {REDUND_UNREPLICABLE} BOOL := FALSE;
		i : {REDUND_UNREPLICABLE} INT;
		LastInformationIndex : {REDUND_UNREPLICABLE} INT;
		LastAnomalyIndex : {REDUND_UNREPLICABLE} INT;
		LastWarningIndex : {REDUND_UNREPLICABLE} INT;
		AuxResetRequired : {REDUND_UNREPLICABLE} BOOL;
		Firstslot : STRING[79];
		Secondslot : STRING[79];
		Thirdslot : STRING[79];
		Fourthslot : STRING[79];
		Fifthslot : STRING[80];
	END_VAR
END_FUNCTION_BLOCK
```

### Program Logical/InputBridge (IEC)

#### InputBridge.st - Cyclic code
```iecst
PROGRAM _CYCLIC

	(*** FEEDER ***)
	LaserSensor1				:= ComTCP_SimInputs.laser_sensor_IR;  (* box present at the end of the first conveyor (conveyor_if) *)
	LaserSensor2 				:= ComTCP_SimInputs.laser_sensor2_IR; (* product passing from conveyor_turn1 towards conveyor_end *)
	Feeder_Carriage_Axis		:= ComTCP_SimInputs.carriage_2_AXIS;  (* actual position of the box group pusher *)
	Feeder_Carriage_Reached		:= ComTCP_SimInputs.carriage_2_RCHD;  (* box group pusher target position reached *)
	Pusher_BKW					:= ComTCP_SimInputs.pusher_LBK;       (* pusher in backward position *)
	Pusher_FWD					:= ComTCP_SimInputs.pusher_LFR; 	  (* pusher in forward position *)
	Turnpusher_BWD				:= ComTCP_SimInputs.turnpusher_LBK;   (* turnpusher in backward position *)
	Turnpusher_FWD				:= ComTCP_SimInputs.turnpusher_LFR;   (* turnpusher in forward position *)

	(*** CRANE ***)
	Crane_Vacuum				:= ComTCP_SimInputs.vaccum_box_crane_VACUUM; (* BOOL vaccum_box_crane_VACUUM *)
	Crane_Box_Axis				:= ComTCP_SimInputs.box_crane_AXIS; 		 (* REAL box_crane_AXIS *)
	Crane_Gantry_Axis			:= ComTCP_SimInputs.gantry_crane_AXIS; 		 (* REAL gantry_crane_AXIS *)

	(*** PALLET ***)
//	Pallet_Fork_EN				:= ComTCP_SimInputs.pallet_fork_left_FB; 		(* BOOL pallet_fork_left_FB *)
	Pallet_ForkFB				:= ComTCP_SimInputs.pallet_fork_left_FB; 		(* BOOL pallet_fork_left_FB *)
	LightBarrier1				:= ComTCP_SimInputs.pallet_light_barrier_1_IR;  (* BOOL pallet_light_barrier_1_IR *)
	LightBarrier2				:= ComTCP_SimInputs.pallet_light_barrier_2_IR;  (* BOOL pallet_light_barrier_2_IR *)
	Pallet_Lifter_Axis			:= ComTCP_SimInputs.pallet_lifter_AXIS; 		(* REAL pallet_lifter_AXIS *)

END_PROGRAM
```

### Program Logical/OutputBridge (IEC)

#### OutputBridge.st - Cyclic code
```iecst
PROGRAM _CYCLIC

	(*** FEEDER ***)
	ComTCP_SimOutputs.conveyor_if_FWD	 := Feeder_ConveyorIF_Fwd; 	 		(* box conveyor (conveyor_if) activation *)
	ComTCP_SimOutputs.conveyer_turn1_FWD := Feeder_ConveyorTurn1_Fwd; 		(* second conveyor activation *)
	ComTCP_SimOutputs.conveyer_end_FWD	 := Feeder_ConveyorEndFwd; 	 		(* third conveyor activation *)
	ComTCP_SimOutputs.pusher_FW			 := Feeder_PusherFwd;				(* pusher activation *)
	ComTCP_SimOutputs.turnpusher_BWD	 := Feeder_TurnpusherBwd; 	 		(* move turnpusher in backward position *)
	ComTCP_SimOutputs.turnpusher_FWD	 := Feeder_TurnpusherFwd; 	 	    (* move turnpusher in forward position *)
	ComTCP_SimOutputs.carriage_2_TGT_POS := Feeder_Carriage_Axis_TgtPos;    (* target position for the box group pusher *)

	(*** CRANE ***)
	ComTCP_SimOutputs.vaccum_box_crane_GRIP	:= Crane_VacuumGrip; 		 	(* BOOL vaccum_box_crane_GRIP *)
	ComTCP_SimOutputs.slide_rail_right_EN	:= Crane_SlideRail_EN; 		 	(* BOOL slide_rail_right_EN *)
	ComTCP_SimOutputs.pusher_x_EN			:= Crane_PusherX_EN; 		 	(* BOOL pusher_x_EN *)
	ComTCP_SimOutputs.pusher_z_EN			:= Crane_PusherZ_EN; 		 	(* BOOL pusher_z_EN *)
	ComTCP_SimOutputs.cartboard_TRIG		:= Crane_CartboardTrig; 	 	(* BOOL cartboard_TRIG *)
	ComTCP_SimOutputs.gantry_crane_TGT_POS	:= Crane_Gantry_Axis_TgtPos; 	(* REAL gantry_crane_TGT_POS *)
	ComTCP_SimOutputs.box_crane_TGT_POS		:= Crane_Box_Axis_TgtPos; 	 	(* REAL box_crane_TGT_POS *)

	(*** PALLET ***)
	ComTCP_SimOutputs.pallet_fork_left_EN		:= Pallet_Fork_EN;			     (* BOOL pallet_fork_left_EN *)
	ComTCP_SimOutputs.pallet_conveyor_1_FWD		:= Pallet_Conveyor1_Fwd; 		 (* BOOL pallet_conveyor_1_FWD *)
	ComTCP_SimOutputs.pallet_conveyor_2_ACT_VEL	:= Pallet_Conveyor2_ActVel;		 (* REAL pallet_conveyor_2_ACT_VEL *)
	ComTCP_SimOutputs.pallet_lifter_TGT_POS		:= Pallet_Lifter_Axis_TgtPos;	 (* REAL pallet_lifter_TGT_POS *)

END_PROGRAM
```

### Program Logical/Feeder (IEC)

#### Feeder.st - Cyclic code
```iecst
PROGRAM _CYCLIC

	CASE State OF

		F_StopSequence:

			StartFeeder						:= FALSE;
			Conveyor_if_disable_request		:= TRUE;
			Conveyor_turn1_disable_request	:= TRUE;
			Conveyor_end_disable_request	:= TRUE;
			Carriage.Command				:= EMERGENCY_STOP_REQUEST;
			State							:= F_StopDONE;

		F_StopDONE:

			IF (NOT Conveyor_if_disable_request AND NOT Conveyor_turn1_disable_request AND NOT Conveyor_end_disable_request AND CarriagePositionReached) THEN
				Carriage.Command		:= IDLE;
				Feeder_EmergencyStop	:= FALSE;
				Feeder_ImmediateStop	:= FALSE;
				Feeder_OnPhaseStop		:= FALSE;
				StopRequest				:= TRUE;
				State					:= F_WaitStart;
			END_IF;

		F_ResetConfig:

			IF NOT Feeder_ResetConfig THEN
				State := F_WaitStart;
			END_IF;

			IF (CarriagePositionReached AND NOT Pusher_disable_request AND NOT Turnpusher_disable_request) THEN
				Carriage.Command	:= IDLE;
				SensorMemory[0]		:= FALSE;
				SensorMemory[1]		:= FALSE;
				SensorReached[0]	:= FALSE;
				SensorReached[1]	:= FALSE;

				FOR i:=0 TO 9 DO
					GD_StatusRequest[i]	:= FALSE;
				END_FOR;

				Feeder_ResetConfig  := FALSE;
				State := F_WaitStart;
			END_IF;

		F_RestoreConfig1:

			Carriage.Command := IDLE;

			FOR i:= 0 TO 9 DO
				IF GD_StatusRequest[i] THEN
					CASE i OF
						0:	Conveyor_if_enable_request		:= TRUE;
						1: 	Conveyor_if_disable_request		:= TRUE;
						2:	Conveyor_turn1_enable_request	:= TRUE;
						3: 	Conveyor_turn1_disable_request	:= TRUE;
						4:	Conveyor_end_enable_request		:= TRUE;
						5:	Conveyor_end_disable_request	:= TRUE;
						6:	Pusher_enable_request			:= TRUE;
						7: 	Pusher_disable_request			:= TRUE;
						8:	Turnpusher_enable_request		:= TRUE;
						9:	Turnpusher_disable_request		:= TRUE;
					END_CASE;
				END_IF;
			END_FOR;

			Enable_Disable_Counter	:= 70;
			State					:= F_RestoreConfig2;

		F_RestoreConfig2:

			FOR i:= 0 TO 9 DO
				IF GD_StatusRequest[i] THEN
					CASE i OF

						0:	IF NOT Conveyor_if_enable_request  THEN
	  							GD_StatusRequest[i]	:= FALSE;
							END_IF;

						1: IF NOT Conveyor_if_disable_request  THEN
								GD_StatusRequest[i]	:= FALSE;
							END_IF;

						2:	IF NOT Conveyor_turn1_enable_request  THEN
								GD_StatusRequest[i]	:= FALSE;
							END_IF;

						3: 	IF NOT Conveyor_turn1_disable_request  THEN
								GD_StatusRequest[i]	:= FALSE;
							END_IF;

						4:	IF NOT Conveyor_end_enable_request  THEN
								GD_StatusRequest[i]	:= FALSE;
							END_IF;

						5:	IF NOT Conveyor_end_disable_request  THEN
								GD_StatusRequest[i]	:= FALSE;
							END_IF;

						6:	IF NOT Pusher_enable_request  THEN
								GD_StatusRequest[i]	:= FALSE;
							END_IF;

						7: 	IF NOT Pusher_disable_request  THEN
								GD_StatusRequest[i]	:= FALSE;
							END_IF;

						8:	IF NOT Turnpusher_enable_request  THEN
								GD_StatusRequest[i]	:= FALSE;
							END_IF;

						9:	IF NOT Turnpusher_disable_request  THEN
								GD_StatusRequest[i]	:= FALSE;
							END_IF;

					END_CASE;
				END_IF;
			END_FOR;

			Enable_Disable_Counter	:= Enable_Disable_Counter - 1;

			IF Enable_Disable_Counter = 0 THEN

				IF CheckPosition THEN
					CarriageSetPoint	:= OldPosition;
					Carriage.Command	:= CHANGE_POSITION;
				END_IF;

				State := F_RestoreConfig3;
			END_IF;

		F_RestoreConfig3:

			IF (CarriagePositionReached AND CheckPosition) THEN
				Carriage.Command			:= IDLE;
				CarriagePositionRestored	:= TRUE;
			END_IF;

			IF (NOT CheckPosition OR CarriagePositionRestored) THEN
				StopRequest		:= FALSE;
				Feeder_Restart	:= FALSE;
				State			:= OldState;
			END_IF;

		F_WaitStart:

			IF Feeder_Restart THEN
				State := F_RestoreConfig1;
			END_IF;

			IF Feeder_ResetConfig THEN
				BoxCounter					:= 0;
				FeederReady					:= FALSE;
				CraneLayerCounter			:= FALSE;
				SecondLayer					:= FALSE;
				LoadBoxesOnCrane			:= FALSE;
				BoxesOnCrane				:= FALSE;
				Pusher_disable_request		:= TRUE;
				Turnpusher_disable_request	:= TRUE;
				CarriageSetPoint			:= 0;
				Carriage.Command			:= CHANGE_POSITION;
				State						:= F_ResetConfig;
			END_IF;

			IF (StartFeeder AND NOT Feeder_ResetConfig AND NOT Feeder_Restart) THEN
				Conveyor_if_enable_request	:= TRUE;
				State						:= F_WaitConveyorIFActive;
			END_IF;

			IF Feeder_EmergencyStop THEN
	  			State := F_StopSequence;
			END_IF;

			IF Feeder_ImmediateStop AND NOT StopRequest THEN
				OldState := State;
				State	 := F_StopSequence;
			END_IF;

			IF Feeder_ImmediateStop AND StopRequest THEN
				State	:= F_StopSequence;
			END_IF;

		F_WaitConveyorIFActive:

			IF NOT Conveyor_if_enable_request THEN
				State	:= F_WaitBoxPusherPosition;
			END_IF;

			IF Feeder_EmergencyStop THEN
				State	:= F_StopSequence;
			END_IF;

			IF Feeder_ImmediateStop THEN
				GD_StatusRequest[0]		  := TRUE; (* conveyor_if_EN *)
				OldState				  := State;
				State				   	  := F_StopSequence;
			END_IF;

		F_WaitBoxPusherPosition:

			IF (LaserSensor1 OR (SensorReached[0] AND SensorMemory[0])) THEN
				SensorReached[0]				:= FALSE;
				SensorMemory[0]					:= FALSE;
				Conveyor_if_disable_request		:= TRUE;
				Conveyor_turn1_enable_request	:= TRUE;
				Conveyor_end_enable_request		:= TRUE;
				State							:= F_LayerCheck;
			END_IF;

			IF Feeder_EmergencyStop THEN
				State	:= F_StopSequence;
			END_IF;

			IF Feeder_ImmediateStop THEN
				SensorMemory[0]			  := TRUE; (* laser_sensor_IR *)
				GD_StatusRequest[0] 	  := TRUE; (* conveyor_if_EN *)
				OldState				  := State;
				State					  := F_StopSequence;
			END_IF;

		F_LayerCheck:

			IF (NOT Conveyor_if_disable_request AND NOT Conveyor_turn1_enable_request AND NOT Conveyor_end_enable_request) THEN

				IF NOT CraneLayerCounter THEN		(* 1st boxes layer *)
					IF BoxCounter < 8 THEN
						Turnpusher_disable_request	:= TRUE;
						Pusher_enable_request		:= TRUE;
						MainLine					:= TRUE;
						State						:= F_LineCheck;
					END_IF;

					IF BoxCounter >= 8 THEN
						Turnpusher_enable_request	:= TRUE;
						Pusher_enable_request	    := TRUE;
						MainLine					:= FALSE;
						State						:= F_LineCheck;
					END_IF;
				END_IF;

				IF CraneLayerCounter THEN		(* 2nd boxes layer *)
					IF BoxCounter < 6 THEN
						Turnpusher_enable_request	:= TRUE;
						Pusher_enable_request		:= TRUE;
						MainLine					:= FALSE;
						State						:= F_LineCheck;
					END_IF;

					IF BoxCounter >= 6 THEN
						Turnpusher_disable_request	:= TRUE;
						Pusher_enable_request		:= TRUE;
						MainLine					:= TRUE;
						State						:= F_LineCheck;
					END_IF;
				END_IF;

			END_IF;

			IF Feeder_EmergencyStop THEN
				State	:= F_StopSequence;
			END_IF;

			IF Feeder_ImmediateStop THEN
				GD_StatusRequest[1]	:= TRUE; (* conveyor_if_DIS *)
				GD_StatusRequest[2]	:= TRUE; (* conveyor_turn1_EN *)
				GD_StatusRequest[4]	:= TRUE; (* conveyor_end_EN *)
				OldState			:= State;
				State				:= F_StopSequence;
			END_IF;

		F_LineCheck:

			IF (NOT Turnpusher_disable_request AND NOT Pusher_enable_request AND MainLine) THEN
				Pusher_disable_request	:= TRUE;
				State					:= F_WaitLaser2;
			END_IF;

			IF (NOT Turnpusher_enable_request AND NOT Pusher_enable_request AND NOT MainLine) THEN
				Pusher_disable_request	:= TRUE;
				State					:= F_WaitLaser2;
			END_IF;

			IF Feeder_EmergencyStop THEN
				State	:= F_StopSequence;
			END_IF;

			IF Feeder_ImmediateStop THEN
				SensorMemory[1]		:= TRUE;
				GD_StatusRequest[2]	:= TRUE; (* conveyor_turn1_EN *)
				GD_StatusRequest[4]	:= TRUE; (* conveyor_end_EN *)
				GD_StatusRequest[6]	:= TRUE; (* pusher_EN *)

				IF MainLine THEN
					GD_StatusRequest[9]	:= TRUE; (* turnpusher_DIS *)
				END_IF;
				IF NOT MainLine THEN
					GD_StatusRequest[8]	:= TRUE; (* turnpusher_EN *)
				END_IF;

				OldState	:= State;
				State		:= F_StopSequence;
			END_IF;

		F_WaitLaser2:

			IF ((LaserSensor2 OR (SensorReached[1] AND SensorMemory[1])) AND NOT Pusher_disable_request) THEN
				SensorReached[1]	:= FALSE;
				SensorMemory[1]		:= FALSE;
				BoxCounter			:= BoxCounter + 1;
				State				:= F_BoxPosOk;
			END_IF;

			IF Feeder_EmergencyStop THEN
				State	:= F_StopSequence;
			END_IF;

			IF Feeder_ImmediateStop THEN
				SensorMemory[1]		:= TRUE;
				GD_StatusRequest[2]	:= TRUE; (* conveyor_turn1_EN *)
				GD_StatusRequest[4]	:= TRUE; (* conveyor_end_EN *)
				GD_StatusRequest[7]	:= TRUE; (* pusher_DIS *)
				OldState			:= State;
				State				:= F_StopSequence;
			END_IF;

		F_BoxPosOk:

			IF NOT CraneLayerCounter THEN		(* 1st boxes layer *)

				IF (BoxCounter = 8 OR BoxCounter = 11 OR BoxCounter = 14) THEN
					Conveyor_turn1_disable_request	:= TRUE;
					State							:= F_WaitConveyorStop;
				ELSE
					State							:= F_WaitStart;
				END_IF;

			END_IF;

			IF CraneLayerCounter THEN		(* 2nd boxes layer *)

				IF (BoxCounter = 3 OR BoxCounter = 6 OR BoxCounter = 14) THEN
					Conveyor_turn1_disable_request	:= TRUE;
					State							:= F_WaitConveyorStop;
				ELSE
					State							:= F_WaitStart;
				END_IF;

			END_IF;

			IF Feeder_EmergencyStop THEN
				State	:= F_StopSequence;
			END_IF;

			IF Feeder_ImmediateStop THEN
				GD_StatusRequest[2]	:= TRUE; (* conveyor_turn1_EN *)
				GD_StatusRequest[4]	:= TRUE; (* conveyor_end_EN *)
				OldState			:= State;
				State				:= F_StopSequence;
			END_IF;

		F_WaitConveyorStop:

			IF NOT Conveyor_turn1_disable_request THEN

				IF BoxCounter = 14 THEN
					State	:= F_Idle;
				END_IF;

				IF BoxCounter < 14 THEN
					EndLayer			:= FALSE;
					CarriageSetPoint	:= 0.44;
					Carriage.Command	:= CHANGE_POSITION;
					State				:= F_CarriageFwdPosition;
				END_IF;

			END_IF;

			IF Feeder_EmergencyStop THEN
				State	:= F_StopSequence;
			END_IF;

			IF Feeder_ImmediateStop THEN
				GD_StatusRequest[4]	:= TRUE; (* conveyor_end_EN *)
				GD_StatusRequest[3]	:= TRUE; (* conveyor_turn1_DIS *)
				OldState			:= State;
				State				:= F_StopSequence;
			END_IF;

		F_Idle:

			FeederReady	:= TRUE;

			IF CraneLayerCounter THEN		(* 2nd boxes layer *)
				SecondLayer	:= TRUE;
			END_IF;

			IF LoadBoxesOnCrane THEN
				EndLayer			:= TRUE;
				CraneLayerCounter	:= NOT CraneLayerCounter;
				CarriageSetPoint	:= 1.1;
				Carriage.Command	:= CHANGE_POSITION;		(* Axis command *)
				State				:= F_CarriageFwdPosition;
			END_IF;

			IF Feeder_EmergencyStop THEN
				State	:= F_StopSequence;
			END_IF;

			IF Feeder_ImmediateStop OR Feeder_OnPhaseStop THEN
				GD_StatusRequest[4]	:= TRUE; (* conveyor_end_EN *)
				OldState			:= State;
				State				:= F_StopSequence;
			END_IF;

		F_CarriageFwdPosition:

			IF (CarriagePositionReached OR CarriagePositionRestored) THEN
				CheckPosition			 := FALSE;
				CarriagePositionRestored := FALSE;
				Carriage.Command		 := IDLE;	(* Axis command *)
				State					 := F_CarriageBwdPosition;
			END_IF;

			IF Feeder_EmergencyStop THEN
				State	:= F_StopSequence;
			END_IF;

			IF Feeder_ImmediateStop THEN
				GD_StatusRequest[4]	:= TRUE; (* conveyor_end_EN *)

				IF EndLayer THEN
					CheckPosition	:= TRUE;
					OldPosition		:= 1.1;  (* old carriage position *)
				END_IF;
				IF NOT EndLayer THEN
					CheckPosition	:= TRUE;
					OldPosition		:= 0.44; (* old carriage position *)
				END_IF;

				OldState	:= State;
				State		:= F_StopSequence;
			END_IF;

		F_CarriageBwdPosition:

			IF 	NOT Carriage.InPosition THEN
				CarriageSetPoint	:= 0.0;
				Carriage.Command	:= CHANGE_POSITION;
				State				:= F_WaitStartPosition;
			END_IF;

			IF Feeder_EmergencyStop THEN
				State	:= F_StopSequence;
			END_IF;

			IF Feeder_ImmediateStop THEN
				GD_StatusRequest[4]	:= TRUE; (* conveyor_end_EN *)
				OldState			:= State;
				State				:= F_StopSequence;
			END_IF;

		F_WaitStartPosition:

			IF BoxCounter = 14 THEN
				BoxesOnCrane	:= TRUE;
				BoxCounter		:= 0;
			END_IF;

			IF (CarriagePositionReached OR CarriagePositionRestored) THEN
				CheckPosition		      := FALSE;
				CarriagePositionRestored  := FALSE;
				Carriage.Command		  := IDLE;
				State					  := F_WaitStart;
			END_IF;

			IF Feeder_EmergencyStop THEN
				State	:= F_StopSequence;
			END_IF;

			IF Feeder_ImmediateStop THEN
				GD_StatusRequest[4]  := TRUE; (* conveyor_end_EN *)
				CheckPosition		 := TRUE;
				OldPosition			 := 0; 	(* old carriage position *)
				OldState			 := State;
				State				 := F_StopSequence;
			END_IF;

	END_CASE;

	IF LaserSensor1 THEN
		SensorReached[0]	:= TRUE;
	END_IF;

	IF LaserSensor2 THEN
		SensorReached[1]	:= TRUE;
	END_IF;

	(*** Generic Devices ***)

	Conveyor_if.DeviceOperation 		 := OperationType;
	Conveyor_if.DeviceClock 			 := TRUE;
	Conveyor_if.DeviceDiagnosticsEnabled := TRUE;
	Conveyor_if.DeviceEnablePreset 		 := FALSE;
	Conveyor_if.DeviceEnableTime 		 := Conveyor_if_EnableTime;
	Conveyor_if.DeviceDisableTime 		 := Conveyor_if_DisableTime;
	Conveyor_if.DeviceType 				 := DEVICE_WITHOUT_FEEDBACK OR DEVICE_WITH_SINGLE_ACTUATION;
	Conveyor_if	( DeviceEnableRequest 	 := Conveyor_if_enable_request,
				  DeviceDisableRequest 	 := Conveyor_if_disable_request );
	Feeder_ConveyorIF_Fwd 				 := Conveyor_if.EnableDevice;	(* single actuation *)
	act_ConveyorIFFault					 := SIMConveyorIFFault;

	Conveyor_turn1.DeviceOperation 			:= OperationType;
	Conveyor_turn1.DeviceClock 	   			:= TRUE;
	Conveyor_turn1.DeviceDiagnosticsEnabled := TRUE;
	Conveyor_turn1.DeviceEnablePreset 		:= FALSE;
	Conveyor_turn1.DeviceEnableTime 		:= Conveyor_turn1_EnableTime;
	Conveyor_turn1.DeviceDisableTime 		:= Conveyor_turn1_DisableTime;
	Conveyor_turn1.DeviceType 				:= DEVICE_WITHOUT_FEEDBACK OR DEVICE_WITH_SINGLE_ACTUATION;
	Conveyor_turn1	 ( DeviceEnableRequest  := Conveyor_turn1_enable_request,
					   DeviceDisableRequest := Conveyor_turn1_disable_request );
	Feeder_ConveyorTurn1_Fwd 				:= Conveyor_turn1.EnableDevice;	(* single actuation *)
	act_ConveyorTurn1Fault					:= SIMConveyorTurn1Fault;

	Pusher.DeviceOperation 			:= OperationType;
	Pusher.DeviceClock 				:= TRUE;
	Pusher.DeviceDiagnosticsEnabled := TRUE;
	Pusher.DeviceEnablePreset 		:= FALSE;
	Pusher.DeviceEnabledSensor 		:= Pusher_FWD; (* double feedback *)
	Pusher.DeviceDisabledSensor 	:= Pusher_BKW; (* double feedback *)
	Pusher.DeviceEnableTime 		:= PusherEnableTime;
	Pusher.DeviceDisableTime 		:= PusherDisableTime;
	Pusher.DeviceType 				:= DEVICE_WITH_DOUBLE_FEEDBACK OR DEVICE_WITH_SINGLE_ACTUATION;
	Pusher   ( DeviceEnableRequest  := Pusher_enable_request,
			   DeviceDisableRequest := Pusher_disable_request );
	Feeder_PusherFwd 				:= Pusher.EnableDevice;	(* single actuation *)
	act_FeederPusherFault 			:= SIMFeederPusherFault;

	Conveyor_end.DeviceOperation 			:= OperationType;
	Conveyor_end.DeviceClock 				:= TRUE;
	Conveyor_end.DeviceDiagnosticsEnabled 	:= TRUE;
	Conveyor_end.DeviceEnablePreset 		:= FALSE;
	Conveyor_end.DeviceEnableTime 			:= Conveyor_end_EnableTime;
	Conveyor_end.DeviceDisableTime 			:= Conveyor_end_DisableTime;
	Conveyor_end.DeviceType 				:= DEVICE_WITHOUT_FEEDBACK OR DEVICE_WITH_SINGLE_ACTUATION;
	Conveyor_end     ( DeviceEnableRequest  := Conveyor_end_enable_request,
		               DeviceDisableRequest := Conveyor_end_disable_request );
	Feeder_ConveyorEndFwd 					:= Conveyor_end.EnableDevice;	(* single actuation *)
	act_ConveyorEndFault					:= SIMConveyorEndFault;

	Turnpusher.DeviceOperation 			:= OperationType;
	Turnpusher.DeviceClock 				:= TRUE;
	Turnpusher.DeviceDiagnosticsEnabled := TRUE;
	Turnpusher.DeviceEnablePreset 		:= FALSE;
	Turnpusher.DeviceEnabledSensor 		:= Turnpusher_BWD; (* double feedback *)
	Turnpusher.DeviceDisabledSensor 	:= Turnpusher_FWD; (* double feedback *)
	Turnpusher.DeviceEnableTime 		:= TurnpusherEnableTime;
	Turnpusher.DeviceDisableTime 		:= TurnpusherDisableTime;
	Turnpusher.DeviceType 				:= DEVICE_WITH_DOUBLE_FEEDBACK OR DEVICE_WITH_DOUBLE_ACTUATION;
	Turnpusher   ( DeviceEnableRequest  := Turnpusher_enable_request,
		           DeviceDisableRequest := Turnpusher_disable_request );
	Feeder_TurnpusherBwd 				:= Turnpusher.EnableDevice;		(* double actuation *)
	Feeder_TurnpusherFwd 				:= Turnpusher.DisableDevice;	(* double actuation *)
	act_TurnpusherFault 				:= SIMTurnpusherFault;

	(*** Generic Axis ***)

	Carriage.NewSetPoint		:= CarriageSetPoint;
	Carriage.ActualPosition		:= Feeder_Carriage_Axis;
	Carriage.TGT_SENSOR			:= Feeder_Carriage_Reached;
	Feeder_Carriage_Axis_TgtPos	:= Carriage.TargetPosition;
	CarriagePositionReached		:= Carriage.InPosition;
	Carriage.DeviceTimer		:= 400;
	act_CarriageFault			:= SIMCarriageFault;
	Carriage();

END_PROGRAM
```

#### Types.typ - Local data types
```iecst
TYPE
	FeederState :
		(
		F_StopSequence := 1,
		F_StopDONE := 2,
		F_ResetConfig := 3,
		F_RestoreConfig1 := 4,
		F_RestoreConfig2 := 5,
		F_RestoreConfig3 := 6,
		F_WaitStart := 7,
		F_WaitConveyorIFActive := 8,
		F_WaitBoxPusherPosition := 9,
		F_LayerCheck := 10,
		F_LineCheck := 11,
		F_WaitLaser2 := 12,
		F_BoxPosOk := 13,
		F_WaitConveyorStop := 14,
		F_Idle := 15,
		F_CarriageFwdPosition := 16,
		F_CarriageBwdPosition := 17,
		F_WaitStartPosition := 18
		);
END_TYPE
```

#### Variables.var - Local variables
```iecst
VAR
	State : FeederState := F_WaitStart;
END_VAR
(*Conveyor_if*)
VAR
	Conveyor_if : GenericDevice;
	Conveyor_if_EnableTime : INT := 20;
	Conveyor_if_DisableTime : INT := 20;
END_VAR
(*Conveyor_turn1*)
VAR
	Conveyor_turn1 : GenericDevice;
	Conveyor_turn1_EnableTime : INT := 20;
	Conveyor_turn1_DisableTime : INT := 20;
END_VAR
(*Pusher*)
VAR
	Pusher : GenericDevice;
	PusherEnableTime : INT := 60;
	PusherDisableTime : INT := 60;
END_VAR
(*Conveyor_end*)
VAR
	Conveyor_end : GenericDevice;
	Conveyor_end_EnableTime : INT := 20;
	Conveyor_end_DisableTime : INT := 20;
END_VAR
(*Turnpusher*)
VAR
	Turnpusher : GenericDevice;
	TurnpusherEnableTime : INT := 60;
	TurnpusherDisableTime : INT := 60;
END_VAR
(*Carriage*)
VAR
	Carriage : GenericAxis;
	CarriagePositionReached : BOOL;
	CarriageSetPoint : REAL;
	MainLine : BOOL := FALSE;
END_VAR
(*Faults*)
VAR
	OldState : FeederState;
	GD_StatusRequest : ARRAY[0..9] OF BOOL := [10(FALSE)];
	OldPosition : REAL;
	i : INT := 0;
	EndLayer : BOOL := FALSE;
	Enable_Disable_Counter : INT;
	SensorReached : ARRAY[0..1] OF BOOL := [2(FALSE)];
	CarriagePositionRestored : BOOL := FALSE;
	CheckPosition : BOOL := FALSE;
	SensorMemory : ARRAY[0..1] OF BOOL := [2(FALSE)];
	StopRequest : BOOL := FALSE;
END_VAR
```

### Program Logical/Crane (IEC)
